REGION Network 2: Перше слово повідомлень
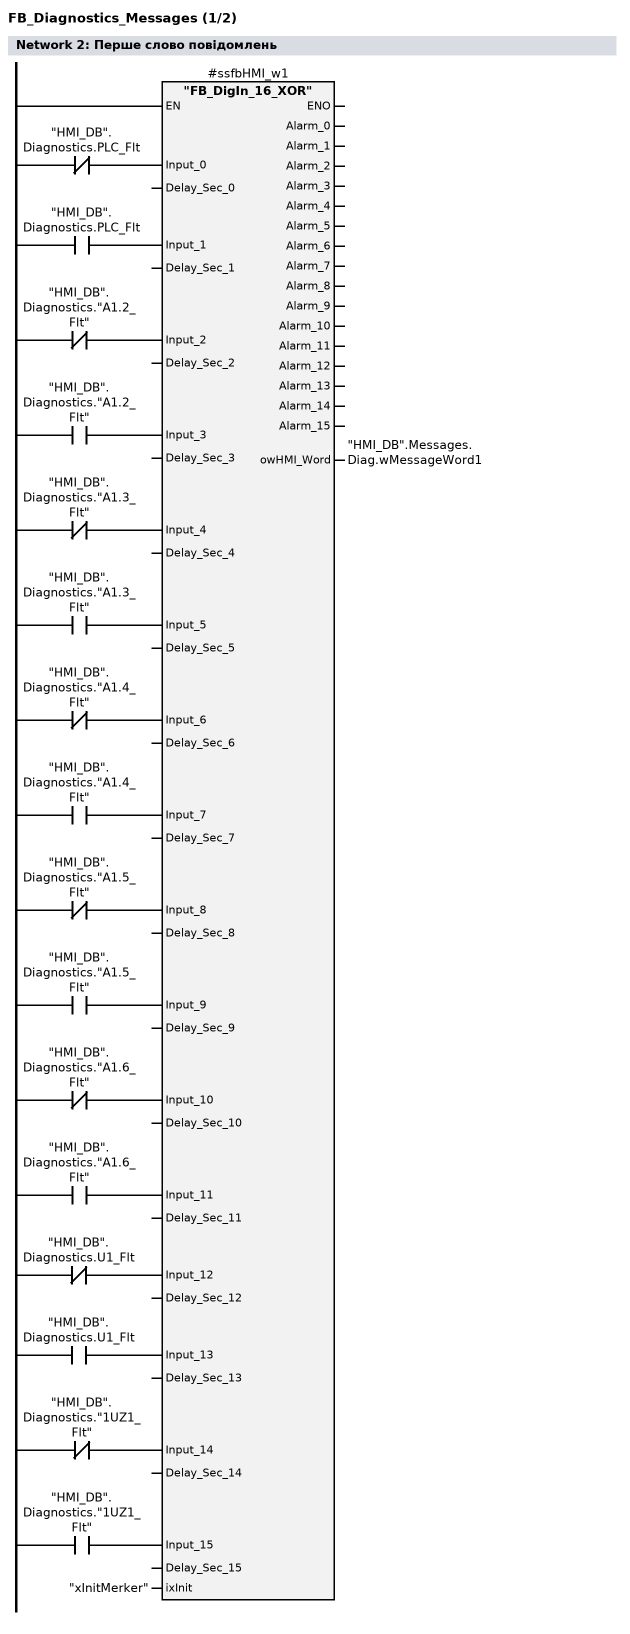
   RUNG wire#powerrail
      #ssfbHMI_w1(Input_0 := wire#w1, Input_1 := wire#w2, Input_2 := wire#w3, Input_3 := wire#w4, Input_4 := wire#w5, Input_5 := wire#w6, Input_6 := wire#w7, Input_7 := wire#w8, Input_8 := wire#w9, Input_9 := wire#w10, Input_10 := wire#w11, Input_11 := wire#w12, Input_12 := wire#w13, Input_13 := wire#w14, Input_14 := wire#w15, Input_15 := wire#w16, Delay_Sec_0 :=, Delay_Sec_1 :=, Delay_Sec_2 :=, Delay_Sec_3 :=, Delay_Sec_4 :=, Delay_Sec_5 :=, Delay_Sec_6 :=, Delay_Sec_7 :=, Delay_Sec_8 :=, Delay_Sec_9 :=, Delay_Sec_10 :=, Delay_Sec_11 :=, Delay_Sec_12 :=, Delay_Sec_13 :=, Delay_Sec_14 :=, Delay_Sec_15 :=, ixInit := "xInitMerker", Alarm_0 =>, Alarm_1 =>, Alarm_2 =>, Alarm_3 =>, Alarm_4 =>, Alarm_5 =>, Alarm_6 =>, Alarm_7 =>, Alarm_8 =>, Alarm_9 =>, Alarm_10 =>, Alarm_11 =>, Alarm_12 =>, Alarm_13 =>, Alarm_14 =>, Alarm_15 =>, owHMI_Word => "HMI_DB".Messages.Diag.wMessageWord1)
   END_RUNG
   RUNG wire#powerrail
      I_Contact( "HMI_DB".Diagnostics.PLC_Flt )
   END_RUNG wire#w1
   RUNG wire#powerrail
      Contact( "HMI_DB".Diagnostics.PLC_Flt )
   END_RUNG wire#w2
   RUNG wire#powerrail
      I_Contact( "HMI_DB".Diagnostics."A1.2_Flt" )
   END_RUNG wire#w3
   RUNG wire#powerrail
      Contact( "HMI_DB".Diagnostics."A1.2_Flt" )
   END_RUNG wire#w4
   RUNG wire#powerrail
      I_Contact( "HMI_DB".Diagnostics."A1.3_Flt" )
   END_RUNG wire#w5
   RUNG wire#powerrail
      Contact( "HMI_DB".Diagnostics."A1.3_Flt" )
   END_RUNG wire#w6
   RUNG wire#powerrail
      I_Contact( "HMI_DB".Diagnostics."A1.4_Flt" )
   END_RUNG wire#w7
   RUNG wire#powerrail
      Contact( "HMI_DB".Diagnostics."A1.4_Flt" )
   END_RUNG wire#w8
   RUNG wire#powerrail
      I_Contact( "HMI_DB".Diagnostics."A1.5_Flt" )
   END_RUNG wire#w9
   RUNG wire#powerrail
      Contact( "HMI_DB".Diagnostics."A1.5_Flt" )
   END_RUNG wire#w10
   RUNG wire#powerrail
      I_Contact( "HMI_DB".Diagnostics."A1.6_Flt" )
   END_RUNG wire#w11
   RUNG wire#powerrail
      Contact( "HMI_DB".Diagnostics."A1.6_Flt" )
   END_RUNG wire#w12
   RUNG wire#powerrail
      I_Contact( "HMI_DB".Diagnostics.U1_Flt )
   END_RUNG wire#w13
   RUNG wire#powerrail
      Contact( "HMI_DB".Diagnostics.U1_Flt )
   END_RUNG wire#w14
   RUNG wire#powerrail
      I_Contact( "HMI_DB".Diagnostics."1UZ1_Flt" )
   END_RUNG wire#w15
   RUNG wire#powerrail
      Contact( "HMI_DB".Diagnostics."1UZ1_Flt" )
   END_RUNG wire#w16
   // the same network as SCL:
   #ssfbHMI_w1(Input_0 := NOT "HMI_DB".Diagnostics.PLC_Flt,   // "FB_DigIn_16_XOR"
               Input_1 := "HMI_DB".Diagnostics.PLC_Flt,
               Input_2 := NOT "HMI_DB".Diagnostics."A1.2_Flt",
               Input_3 := "HMI_DB".Diagnostics."A1.2_Flt",
               Input_4 := NOT "HMI_DB".Diagnostics."A1.3_Flt",
               Input_5 := "HMI_DB".Diagnostics."A1.3_Flt",
               Input_6 := NOT "HMI_DB".Diagnostics."A1.4_Flt",
               Input_7 := "HMI_DB".Diagnostics."A1.4_Flt",
               Input_8 := NOT "HMI_DB".Diagnostics."A1.5_Flt",
               Input_9 := "HMI_DB".Diagnostics."A1.5_Flt",
               Input_10 := NOT "HMI_DB".Diagnostics."A1.6_Flt",
               Input_11 := "HMI_DB".Diagnostics."A1.6_Flt",
               Input_12 := NOT "HMI_DB".Diagnostics.U1_Flt,
               Input_13 := "HMI_DB".Diagnostics.U1_Flt,
               Input_14 := NOT "HMI_DB".Diagnostics."1UZ1_Flt",
               Input_15 := "HMI_DB".Diagnostics."1UZ1_Flt",
               ixInit := "xInitMerker",
               owHMI_Word => "HMI_DB".Messages.Diag.wMessageWord1);
END_REGION

REGION Network 3: Друге слово повідомлень
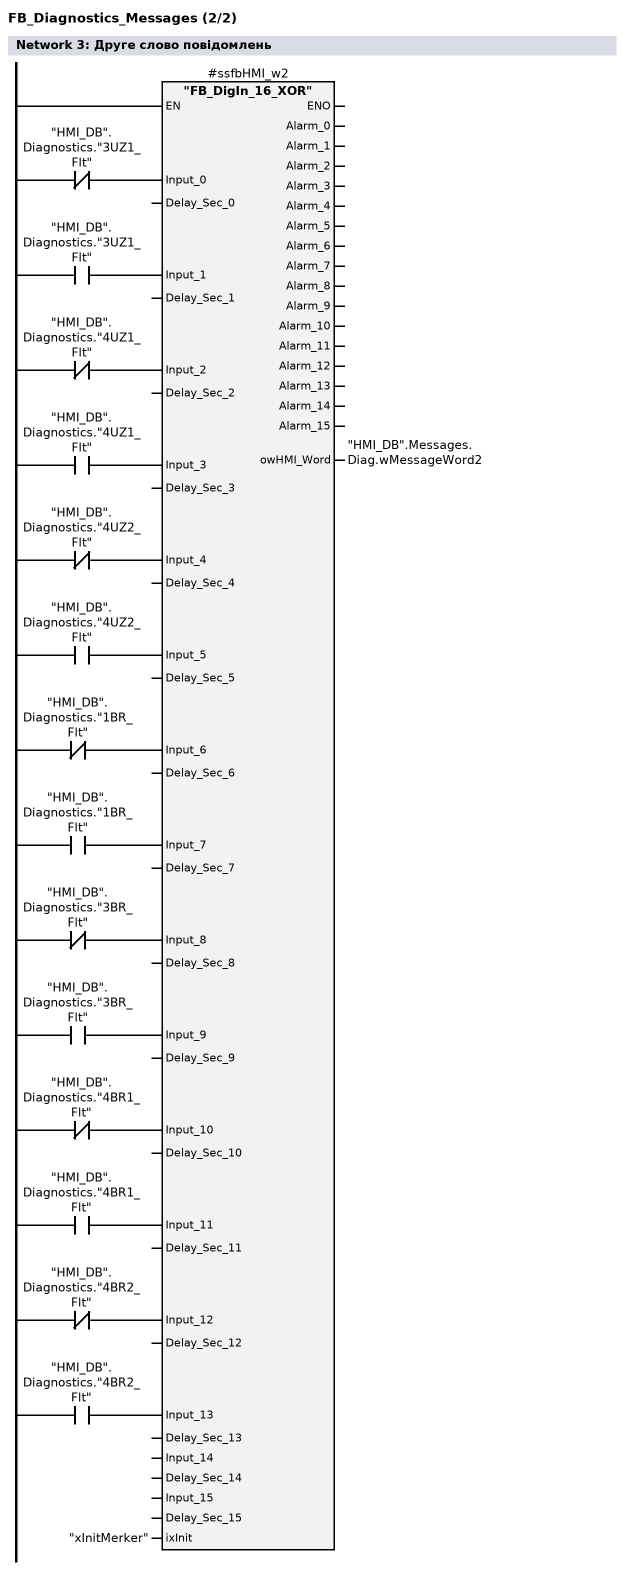
   RUNG wire#powerrail
      #ssfbHMI_w2(Input_0 := wire#w1, Input_1 := wire#w2, Input_2 := wire#w3, Input_3 := wire#w4, Input_4 := wire#w5, Input_5 := wire#w6, Input_6 := wire#w7, Input_7 := wire#w8, Input_8 := wire#w9, Input_9 := wire#w10, Input_10 := wire#w11, Input_11 := wire#w12, Input_12 := wire#w13, Input_13 := wire#w14, Delay_Sec_0 :=, Delay_Sec_1 :=, Delay_Sec_2 :=, Delay_Sec_3 :=, Delay_Sec_4 :=, Delay_Sec_5 :=, Delay_Sec_6 :=, Delay_Sec_7 :=, Delay_Sec_8 :=, Delay_Sec_9 :=, Delay_Sec_10 :=, Delay_Sec_11 :=, Delay_Sec_12 :=, Delay_Sec_13 :=, Input_14 :=, Delay_Sec_14 :=, Input_15 :=, Delay_Sec_15 :=, ixInit := "xInitMerker", Alarm_0 =>, Alarm_1 =>, Alarm_2 =>, Alarm_3 =>, Alarm_4 =>, Alarm_5 =>, Alarm_6 =>, Alarm_7 =>, Alarm_8 =>, Alarm_9 =>, Alarm_10 =>, Alarm_11 =>, Alarm_12 =>, Alarm_13 =>, Alarm_14 =>, Alarm_15 =>, owHMI_Word => "HMI_DB".Messages.Diag.wMessageWord2)
   END_RUNG
   RUNG wire#powerrail
      I_Contact( "HMI_DB".Diagnostics."3UZ1_Flt" )
   END_RUNG wire#w1
   RUNG wire#powerrail
      Contact( "HMI_DB".Diagnostics."3UZ1_Flt" )
   END_RUNG wire#w2
   RUNG wire#powerrail
      I_Contact( "HMI_DB".Diagnostics."4UZ1_Flt" )
   END_RUNG wire#w3
   RUNG wire#powerrail
      Contact( "HMI_DB".Diagnostics."4UZ1_Flt" )
   END_RUNG wire#w4
   RUNG wire#powerrail
      I_Contact( "HMI_DB".Diagnostics."4UZ2_Flt" )
   END_RUNG wire#w5
   RUNG wire#powerrail
      Contact( "HMI_DB".Diagnostics."4UZ2_Flt" )
   END_RUNG wire#w6
   RUNG wire#powerrail
      I_Contact( "HMI_DB".Diagnostics."1BR_Flt" )
   END_RUNG wire#w7
   RUNG wire#powerrail
      Contact( "HMI_DB".Diagnostics."1BR_Flt" )
   END_RUNG wire#w8
   RUNG wire#powerrail
      I_Contact( "HMI_DB".Diagnostics."3BR_Flt" )
   END_RUNG wire#w9
   RUNG wire#powerrail
      Contact( "HMI_DB".Diagnostics."3BR_Flt" )
   END_RUNG wire#w10
   RUNG wire#powerrail
      I_Contact( "HMI_DB".Diagnostics."4BR1_Flt" )
   END_RUNG wire#w11
   RUNG wire#powerrail
      Contact( "HMI_DB".Diagnostics."4BR1_Flt" )
   END_RUNG wire#w12
   RUNG wire#powerrail
      I_Contact( "HMI_DB".Diagnostics."4BR2_Flt" )
   END_RUNG wire#w13
   RUNG wire#powerrail
      Contact( "HMI_DB".Diagnostics."4BR2_Flt" )
   END_RUNG wire#w14
   // the same network as SCL:
   #ssfbHMI_w2(Input_0 := NOT "HMI_DB".Diagnostics."3UZ1_Flt",   // "FB_DigIn_16_XOR"
               Input_1 := "HMI_DB".Diagnostics."3UZ1_Flt",
               Input_2 := NOT "HMI_DB".Diagnostics."4UZ1_Flt",
               Input_3 := "HMI_DB".Diagnostics."4UZ1_Flt",
               Input_4 := NOT "HMI_DB".Diagnostics."4UZ2_Flt",
               Input_5 := "HMI_DB".Diagnostics."4UZ2_Flt",
               Input_6 := NOT "HMI_DB".Diagnostics."1BR_Flt",
               Input_7 := "HMI_DB".Diagnostics."1BR_Flt",
               Input_8 := NOT "HMI_DB".Diagnostics."3BR_Flt",
               Input_9 := "HMI_DB".Diagnostics."3BR_Flt",
               Input_10 := NOT "HMI_DB".Diagnostics."4BR1_Flt",
               Input_11 := "HMI_DB".Diagnostics."4BR1_Flt",
               Input_12 := NOT "HMI_DB".Diagnostics."4BR2_Flt",
               Input_13 := "HMI_DB".Diagnostics."4BR2_Flt",
               ixInit := "xInitMerker",
               owHMI_Word => "HMI_DB".Messages.Diag.wMessageWord2);
END_REGION
END_FUNCTION_BLOCK

FUNCTION "FC_Diagnostic" : Void   // FC600, LAD
{ S7_Optimized_Access := 'TRUE' }
VERSION : 0.1
BEGIN

REGION Network 2: =================ПЛК=======================
END_REGION

REGION Network 3: CPU 1515-2 PN
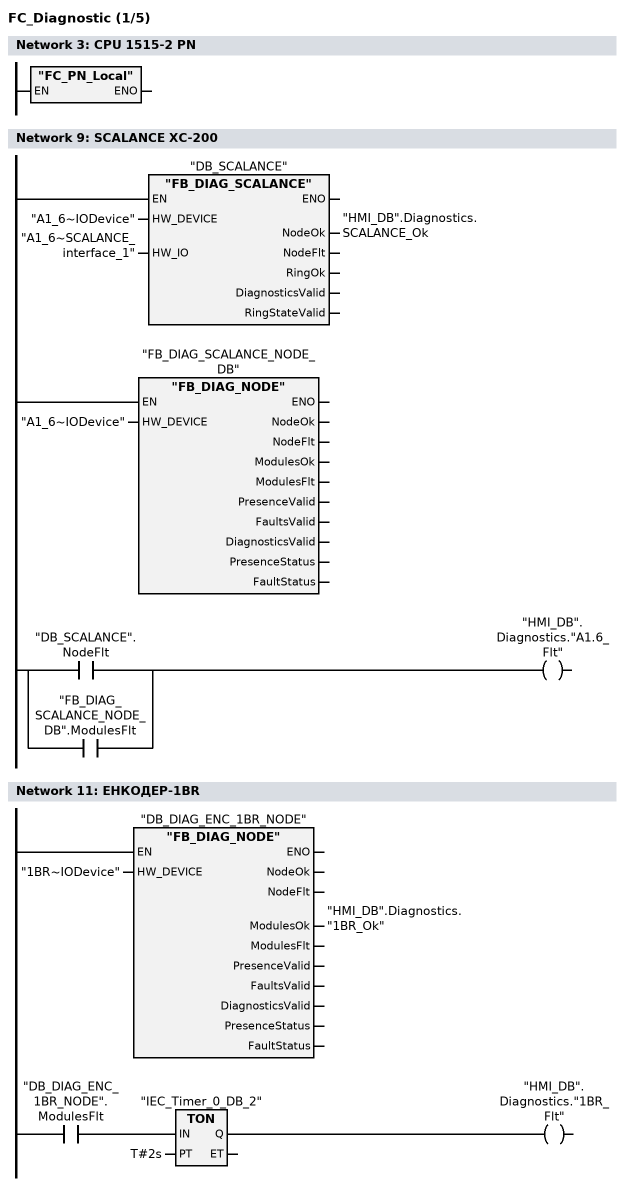
   RUNG wire#powerrail
      "FC_PN_Local"()
   END_RUNG
   // the same network as SCL:
   "FC_PN_Local"();
END_REGION

REGION Network 4: Модуль А1.2
END_REGION

REGION Network 5: Модуль А1.3
END_REGION

REGION Network 6: Модуль А1.4
END_REGION

REGION Network 7: Модуль А1.5
END_REGION

REGION Network 8: =================Мережева діагностіка=======================
END_REGION

REGION Network 9: SCALANCE XC-200
   RUNG wire#powerrail
      "DB_SCALANCE"(HW_DEVICE := "A1_6~IODevice", HW_IO := "A1_6~SCALANCE_interface_1", NodeOk => "HMI_DB".Diagnostics.SCALANCE_Ok, NodeFlt =>, RingOk =>, DiagnosticsValid =>, RingStateValid =>)
   END_RUNG
   RUNG wire#powerrail
      "FB_DIAG_SCALANCE_NODE_DB"(HW_DEVICE := "A1_6~IODevice", NodeOk =>, NodeFlt =>, ModulesOk =>, ModulesFlt =>, PresenceValid =>, FaultsValid =>, DiagnosticsValid =>, PresenceStatus =>, FaultStatus =>)
   END_RUNG
   RUNG wire#powerrail
      Contact( "DB_SCALANCE".NodeFlt )
      wire#w1
      Coil( "HMI_DB".Diagnostics."A1.6_Flt" )
   END_RUNG
   RUNG wire#powerrail
      Contact( "FB_DIAG_SCALANCE_NODE_DB".ModulesFlt )
   END_RUNG wire#w1
   // the same network as SCL:
   "DB_SCALANCE"(HW_DEVICE := "A1_6~IODevice",   // "FB_DIAG_SCALANCE"
                 HW_IO := "A1_6~SCALANCE_interface_1",
                 NodeOk => "HMI_DB".Diagnostics.SCALANCE_Ok);
   "FB_DIAG_SCALANCE_NODE_DB"(HW_DEVICE := "A1_6~IODevice");   // "FB_DIAG_NODE"
   "HMI_DB".Diagnostics."A1.6_Flt" := "DB_SCALANCE".NodeFlt OR "FB_DIAG_SCALANCE_NODE_DB".ModulesFlt;
END_REGION

REGION Network 10: =================Енкодери==================
END_REGION

REGION Network 11: ЕНКОДЕР-1BR
   "DB_DIAG_ENC_1BR_NODE"(HW_DEVICE := "1BR~IODevice", ModulesOk => "HMI_DB".Diagnostics."1BR_Ok");   // "FB_DIAG_NODE"
   "IEC_Timer_0_DB_2".TON(IN := "DB_DIAG_ENC_1BR_NODE".ModulesFlt, PT := T#2s);
   "HMI_DB".Diagnostics."1BR_Flt" := "IEC_Timer_0_DB_2".Q;
END_REGION

REGION Network 12: ЕНКОДЕР-3BR
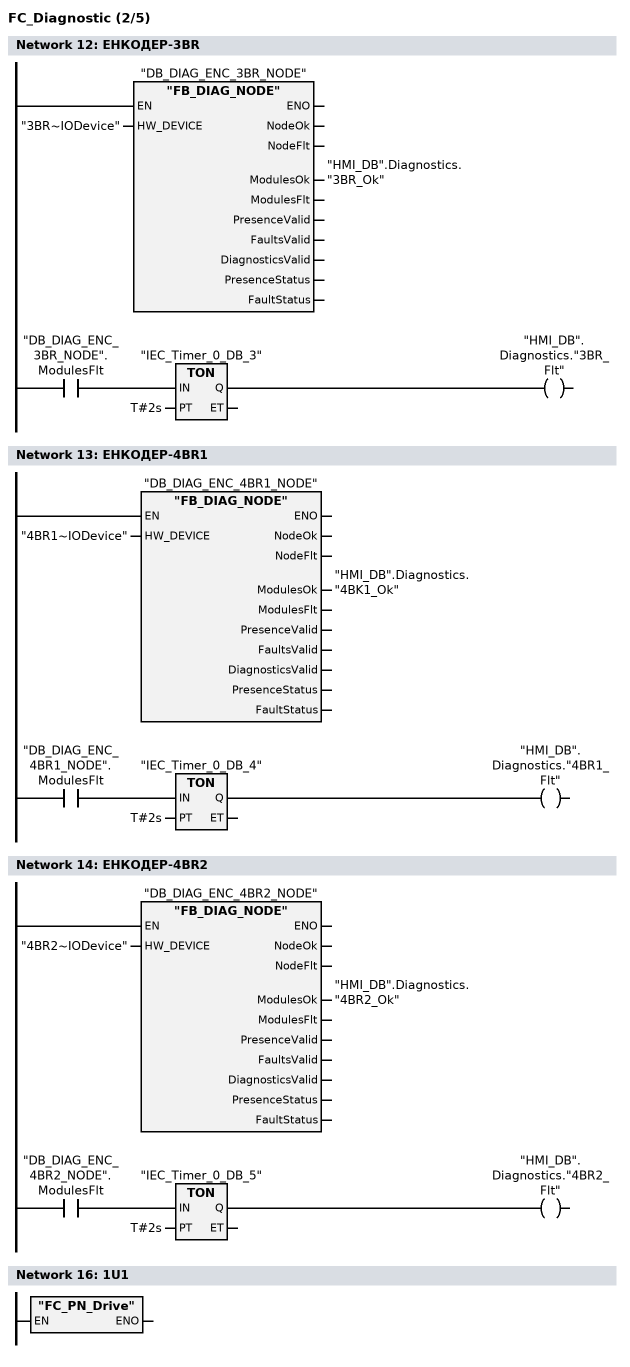
   "DB_DIAG_ENC_3BR_NODE"(HW_DEVICE := "3BR~IODevice", ModulesOk => "HMI_DB".Diagnostics."3BR_Ok");   // "FB_DIAG_NODE"
   "IEC_Timer_0_DB_3".TON(IN := "DB_DIAG_ENC_3BR_NODE".ModulesFlt, PT := T#2s);
   "HMI_DB".Diagnostics."3BR_Flt" := "IEC_Timer_0_DB_3".Q;
END_REGION

REGION Network 13: ЕНКОДЕР-4BR1
   "DB_DIAG_ENC_4BR1_NODE"(HW_DEVICE := "4BR1~IODevice", ModulesOk => "HMI_DB".Diagnostics."4BK1_Ok");   // "FB_DIAG_NODE"
   "IEC_Timer_0_DB_4".TON(IN := "DB_DIAG_ENC_4BR1_NODE".ModulesFlt, PT := T#2s);
   "HMI_DB".Diagnostics."4BR1_Flt" := "IEC_Timer_0_DB_4".Q;
END_REGION

REGION Network 14: ЕНКОДЕР-4BR2
   "DB_DIAG_ENC_4BR2_NODE"(HW_DEVICE := "4BR2~IODevice", ModulesOk => "HMI_DB".Diagnostics."4BR2_Ok");   // "FB_DIAG_NODE"
   "IEC_Timer_0_DB_5".TON(IN := "DB_DIAG_ENC_4BR2_NODE".ModulesFlt, PT := T#2s);
   "HMI_DB".Diagnostics."4BR2_Flt" := "IEC_Timer_0_DB_5".Q;
END_REGION

REGION Network 15: =================ПЧ======================
END_REGION

REGION Network 16: 1U1
   RUNG wire#powerrail
      "FC_PN_Drive"()
   END_RUNG
   // the same network as SCL:
   "FC_PN_Drive"();
END_REGION

REGION Network 17: 1UZ1
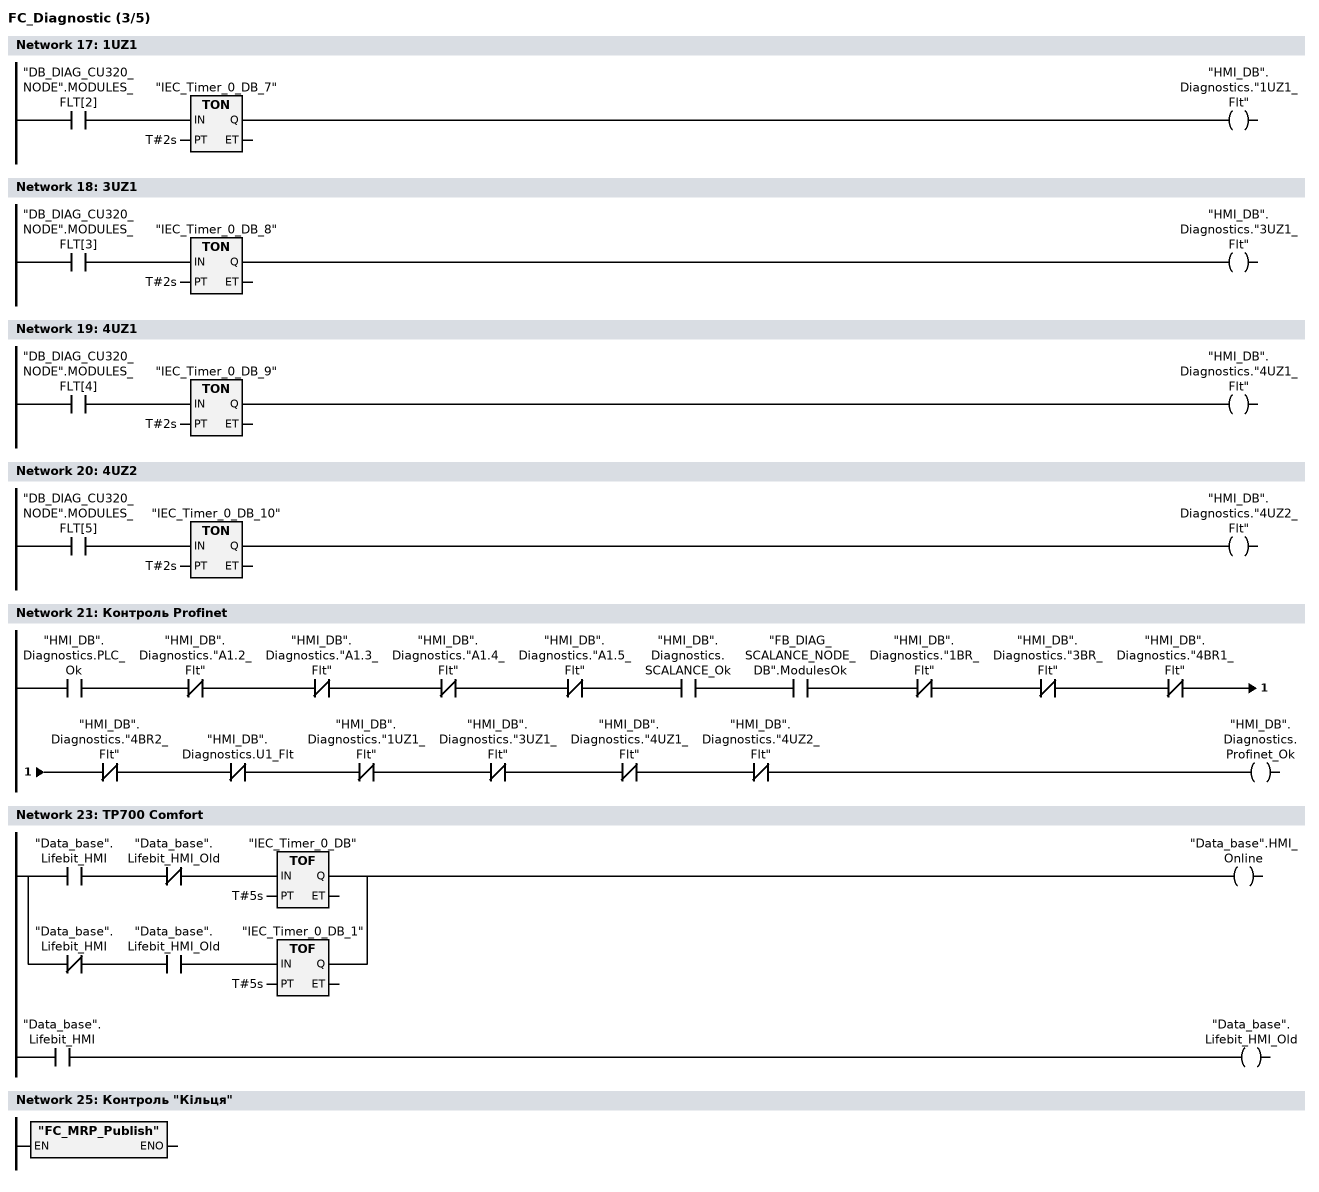
   "IEC_Timer_0_DB_7".TON(IN := "DB_DIAG_CU320_NODE".MODULES_FLT[2], PT := T#2s);
   "HMI_DB".Diagnostics."1UZ1_Flt" := "IEC_Timer_0_DB_7".Q;
END_REGION

REGION Network 18: 3UZ1
   "IEC_Timer_0_DB_8".TON(IN := "DB_DIAG_CU320_NODE".MODULES_FLT[3], PT := T#2s);
   "HMI_DB".Diagnostics."3UZ1_Flt" := "IEC_Timer_0_DB_8".Q;
END_REGION

REGION Network 19: 4UZ1
   "IEC_Timer_0_DB_9".TON(IN := "DB_DIAG_CU320_NODE".MODULES_FLT[4], PT := T#2s);
   "HMI_DB".Diagnostics."4UZ1_Flt" := "IEC_Timer_0_DB_9".Q;
END_REGION

REGION Network 20: 4UZ2
   "IEC_Timer_0_DB_10".TON(IN := "DB_DIAG_CU320_NODE".MODULES_FLT[5], PT := T#2s);
   "HMI_DB".Diagnostics."4UZ2_Flt" := "IEC_Timer_0_DB_10".Q;
END_REGION

REGION Network 21: Контроль Profinet
   RUNG wire#powerrail
      Contact( "HMI_DB".Diagnostics.PLC_Ok )
      I_Contact( "HMI_DB".Diagnostics."A1.2_Flt" )
      I_Contact( "HMI_DB".Diagnostics."A1.3_Flt" )
      I_Contact( "HMI_DB".Diagnostics."A1.4_Flt" )
      I_Contact( "HMI_DB".Diagnostics."A1.5_Flt" )
      Contact( "HMI_DB".Diagnostics.SCALANCE_Ok )
      Contact( "FB_DIAG_SCALANCE_NODE_DB".ModulesOk )
      I_Contact( "HMI_DB".Diagnostics."1BR_Flt" )
      I_Contact( "HMI_DB".Diagnostics."3BR_Flt" )
      I_Contact( "HMI_DB".Diagnostics."4BR1_Flt" )
      I_Contact( "HMI_DB".Diagnostics."4BR2_Flt" )
      I_Contact( "HMI_DB".Diagnostics.U1_Flt )
      I_Contact( "HMI_DB".Diagnostics."1UZ1_Flt" )
      I_Contact( "HMI_DB".Diagnostics."3UZ1_Flt" )
      I_Contact( "HMI_DB".Diagnostics."4UZ1_Flt" )
      I_Contact( "HMI_DB".Diagnostics."4UZ2_Flt" )
      Coil( "HMI_DB".Diagnostics.Profinet_Ok )
   END_RUNG
   // the same network as SCL:
   "HMI_DB".Diagnostics.Profinet_Ok := "HMI_DB".Diagnostics.PLC_Ok AND NOT "HMI_DB".Diagnostics."A1.2_Flt" AND NOT "HMI_DB".Diagnostics."A1.3_Flt" AND NOT "HMI_DB".Diagnostics."A1.4_Flt" AND NOT "HMI_DB".Diagnostics."A1.5_Flt" AND "HMI_DB".Diagnostics.SCALANCE_Ok AND "FB_DIAG_SCALANCE_NODE_DB".ModulesOk AND NOT "HMI_DB".Diagnostics."1BR_Flt" AND NOT "HMI_DB".Diagnostics."3BR_Flt" AND NOT "HMI_DB".Diagnostics."4BR1_Flt" AND NOT "HMI_DB".Diagnostics."4BR2_Flt" AND NOT "HMI_DB".Diagnostics.U1_Flt AND NOT "HMI_DB".Diagnostics."1UZ1_Flt" AND NOT "HMI_DB".Diagnostics."3UZ1_Flt" AND NOT "HMI_DB".Diagnostics."4UZ1_Flt" AND NOT "HMI_DB".Diagnostics."4UZ2_Flt";
END_REGION

REGION Network 22: ================ЛMI======================
END_REGION

REGION Network 23: TP700 Comfort
   "IEC_Timer_0_DB".TOF(IN := "Data_base".Lifebit_HMI AND NOT "Data_base".Lifebit_HMI_Old, PT := T#5s);
   "IEC_Timer_0_DB_1".TOF(IN := NOT "Data_base".Lifebit_HMI AND "Data_base".Lifebit_HMI_Old, PT := T#5s);
   "Data_base".HMI_Online := "IEC_Timer_0_DB".Q OR "IEC_Timer_0_DB_1".Q;
   "Data_base".Lifebit_HMI_Old := "Data_base".Lifebit_HMI;
END_REGION

REGION Network 24: =========================================
END_REGION

REGION Network 25: Контроль "Кільця"
   RUNG wire#powerrail
      "FC_MRP_Publish"()
   END_RUNG
   // the same network as SCL:
   "FC_MRP_Publish"();
END_REGION

REGION Network 26: Формування слова аварій
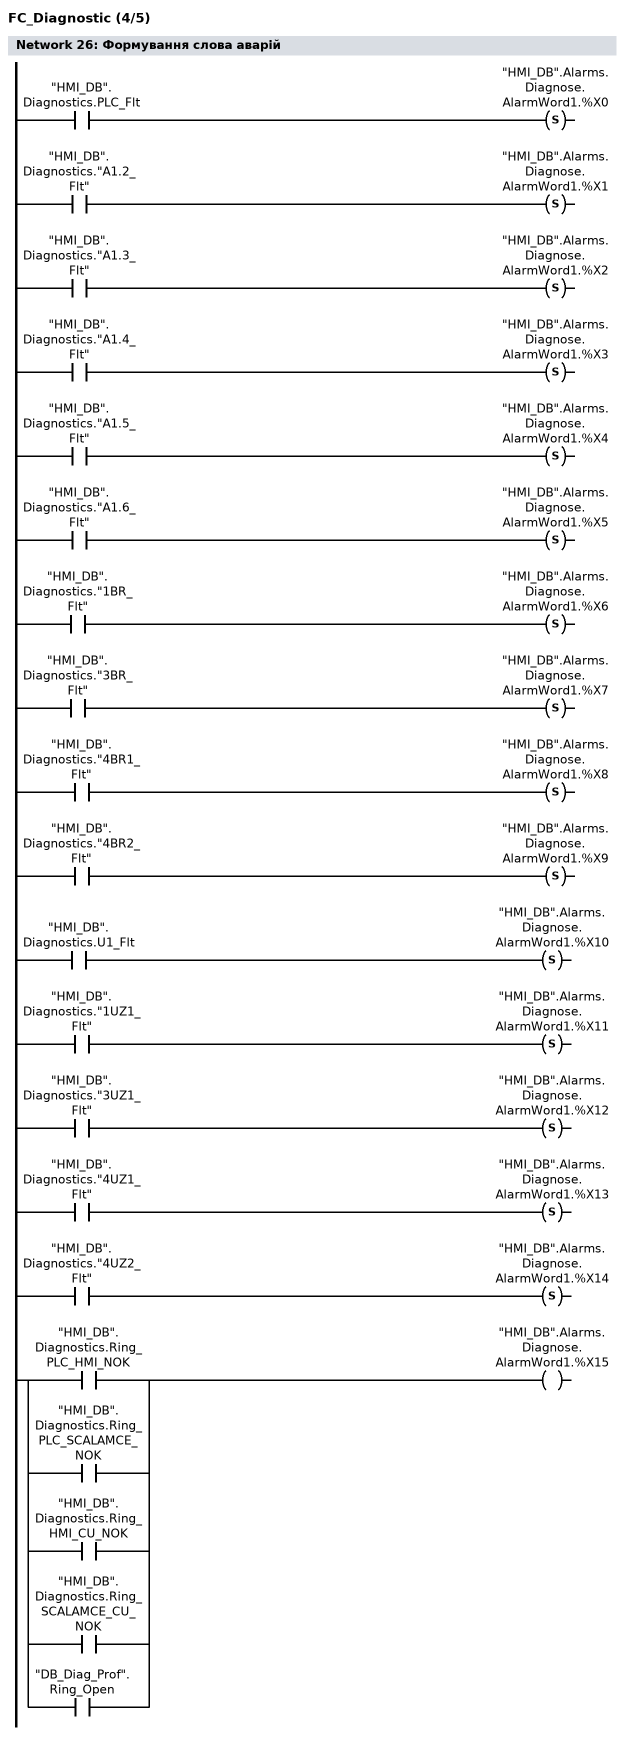
   RUNG wire#powerrail
      Contact( "HMI_DB".Diagnostics.PLC_Flt )
      S_Coil( "HMI_DB".Alarms.Diagnose.AlarmWord1.%X0 )
   END_RUNG
   RUNG wire#powerrail
      Contact( "HMI_DB".Diagnostics."A1.2_Flt" )
      S_Coil( "HMI_DB".Alarms.Diagnose.AlarmWord1.%X1 )
   END_RUNG
   RUNG wire#powerrail
      Contact( "HMI_DB".Diagnostics."A1.3_Flt" )
      S_Coil( "HMI_DB".Alarms.Diagnose.AlarmWord1.%X2 )
   END_RUNG
   RUNG wire#powerrail
      Contact( "HMI_DB".Diagnostics."A1.4_Flt" )
      S_Coil( "HMI_DB".Alarms.Diagnose.AlarmWord1.%X3 )
   END_RUNG
   RUNG wire#powerrail
      Contact( "HMI_DB".Diagnostics."A1.5_Flt" )
      S_Coil( "HMI_DB".Alarms.Diagnose.AlarmWord1.%X4 )
   END_RUNG
   RUNG wire#powerrail
      Contact( "HMI_DB".Diagnostics."A1.6_Flt" )
      S_Coil( "HMI_DB".Alarms.Diagnose.AlarmWord1.%X5 )
   END_RUNG
   RUNG wire#powerrail
      Contact( "HMI_DB".Diagnostics."1BR_Flt" )
      S_Coil( "HMI_DB".Alarms.Diagnose.AlarmWord1.%X6 )
   END_RUNG
   RUNG wire#powerrail
      Contact( "HMI_DB".Diagnostics."3BR_Flt" )
      S_Coil( "HMI_DB".Alarms.Diagnose.AlarmWord1.%X7 )
   END_RUNG
   RUNG wire#powerrail
      Contact( "HMI_DB".Diagnostics."4BR1_Flt" )
      S_Coil( "HMI_DB".Alarms.Diagnose.AlarmWord1.%X8 )
   END_RUNG
   RUNG wire#powerrail
      Contact( "HMI_DB".Diagnostics."4BR2_Flt" )
      S_Coil( "HMI_DB".Alarms.Diagnose.AlarmWord1.%X9 )
   END_RUNG
   RUNG wire#powerrail
      Contact( "HMI_DB".Diagnostics.U1_Flt )
      S_Coil( "HMI_DB".Alarms.Diagnose.AlarmWord1.%X10 )
   END_RUNG
   RUNG wire#powerrail
      Contact( "HMI_DB".Diagnostics."1UZ1_Flt" )
      S_Coil( "HMI_DB".Alarms.Diagnose.AlarmWord1.%X11 )
   END_RUNG
   RUNG wire#powerrail
      Contact( "HMI_DB".Diagnostics."3UZ1_Flt" )
      S_Coil( "HMI_DB".Alarms.Diagnose.AlarmWord1.%X12 )
   END_RUNG
   RUNG wire#powerrail
      Contact( "HMI_DB".Diagnostics."4UZ1_Flt" )
      S_Coil( "HMI_DB".Alarms.Diagnose.AlarmWord1.%X13 )
   END_RUNG
   RUNG wire#powerrail
      Contact( "HMI_DB".Diagnostics."4UZ2_Flt" )
      S_Coil( "HMI_DB".Alarms.Diagnose.AlarmWord1.%X14 )
   END_RUNG
   RUNG wire#powerrail
      Contact( "HMI_DB".Diagnostics.Ring_PLC_HMI_NOK )
      wire#w1
      Coil( "HMI_DB".Alarms.Diagnose.AlarmWord1.%X15 )
   END_RUNG
   RUNG wire#powerrail
      Contact( "HMI_DB".Diagnostics.Ring_PLC_SCALAMCE_NOK )
   END_RUNG wire#w1
   RUNG wire#powerrail
      Contact( "HMI_DB".Diagnostics.Ring_HMI_CU_NOK )
   END_RUNG wire#w1
   RUNG wire#powerrail
      Contact( "HMI_DB".Diagnostics.Ring_SCALAMCE_CU_NOK )
   END_RUNG wire#w1
   RUNG wire#powerrail
      Contact( "DB_Diag_Prof".Ring_Open )
   END_RUNG wire#w1
   // the same network as SCL:
   IF "HMI_DB".Diagnostics.PLC_Flt THEN "HMI_DB".Alarms.Diagnose.AlarmWord1.%X0 := TRUE; END_IF;
   IF "HMI_DB".Diagnostics."A1.2_Flt" THEN "HMI_DB".Alarms.Diagnose.AlarmWord1.%X1 := TRUE; END_IF;
   IF "HMI_DB".Diagnostics."A1.3_Flt" THEN "HMI_DB".Alarms.Diagnose.AlarmWord1.%X2 := TRUE; END_IF;
   IF "HMI_DB".Diagnostics."A1.4_Flt" THEN "HMI_DB".Alarms.Diagnose.AlarmWord1.%X3 := TRUE; END_IF;
   IF "HMI_DB".Diagnostics."A1.5_Flt" THEN "HMI_DB".Alarms.Diagnose.AlarmWord1.%X4 := TRUE; END_IF;
   IF "HMI_DB".Diagnostics."A1.6_Flt" THEN "HMI_DB".Alarms.Diagnose.AlarmWord1.%X5 := TRUE; END_IF;
   IF "HMI_DB".Diagnostics."1BR_Flt" THEN "HMI_DB".Alarms.Diagnose.AlarmWord1.%X6 := TRUE; END_IF;
   IF "HMI_DB".Diagnostics."3BR_Flt" THEN "HMI_DB".Alarms.Diagnose.AlarmWord1.%X7 := TRUE; END_IF;
   IF "HMI_DB".Diagnostics."4BR1_Flt" THEN "HMI_DB".Alarms.Diagnose.AlarmWord1.%X8 := TRUE; END_IF;
   IF "HMI_DB".Diagnostics."4BR2_Flt" THEN "HMI_DB".Alarms.Diagnose.AlarmWord1.%X9 := TRUE; END_IF;
   IF "HMI_DB".Diagnostics.U1_Flt THEN "HMI_DB".Alarms.Diagnose.AlarmWord1.%X10 := TRUE; END_IF;
   IF "HMI_DB".Diagnostics."1UZ1_Flt" THEN "HMI_DB".Alarms.Diagnose.AlarmWord1.%X11 := TRUE; END_IF;
   IF "HMI_DB".Diagnostics."3UZ1_Flt" THEN "HMI_DB".Alarms.Diagnose.AlarmWord1.%X12 := TRUE; END_IF;
   IF "HMI_DB".Diagnostics."4UZ1_Flt" THEN "HMI_DB".Alarms.Diagnose.AlarmWord1.%X13 := TRUE; END_IF;
   IF "HMI_DB".Diagnostics."4UZ2_Flt" THEN "HMI_DB".Alarms.Diagnose.AlarmWord1.%X14 := TRUE; END_IF;
   "HMI_DB".Alarms.Diagnose.AlarmWord1.%X15 := "HMI_DB".Diagnostics.Ring_PLC_HMI_NOK OR "HMI_DB".Diagnostics.Ring_PLC_SCALAMCE_NOK OR "HMI_DB".Diagnostics.Ring_HMI_CU_NOK OR "HMI_DB".Diagnostics.Ring_SCALAMCE_CU_NOK OR "DB_Diag_Prof".Ring_Open;
END_REGION

REGION Network 27: Скидання слова аварій
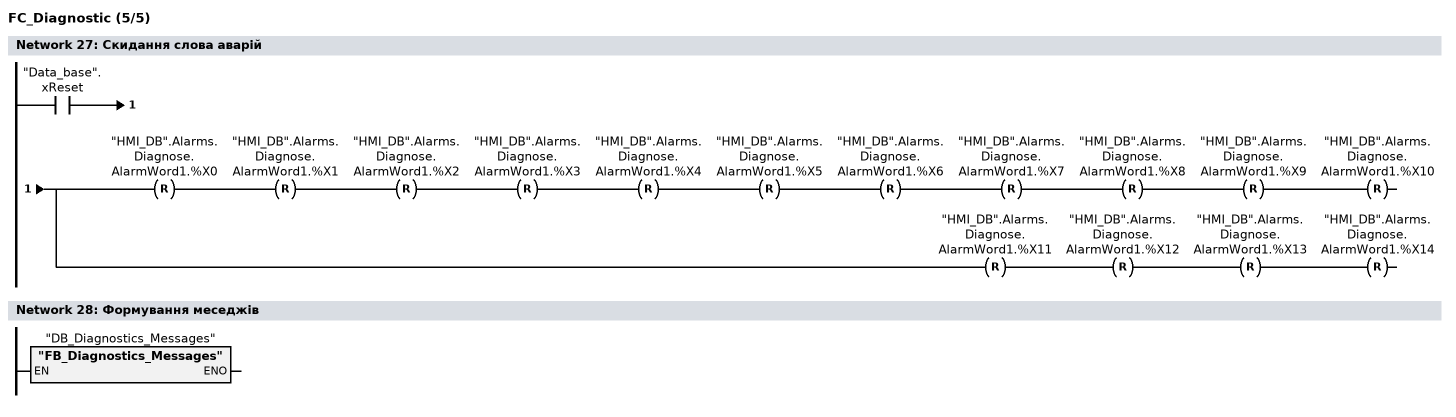
   RUNG wire#powerrail
      Contact( "Data_base".xReset )
      wire#w1
      R_Coil( "HMI_DB".Alarms.Diagnose.AlarmWord1.%X0 )
      R_Coil( "HMI_DB".Alarms.Diagnose.AlarmWord1.%X1 )
      R_Coil( "HMI_DB".Alarms.Diagnose.AlarmWord1.%X2 )
      R_Coil( "HMI_DB".Alarms.Diagnose.AlarmWord1.%X3 )
      R_Coil( "HMI_DB".Alarms.Diagnose.AlarmWord1.%X4 )
      R_Coil( "HMI_DB".Alarms.Diagnose.AlarmWord1.%X5 )
      R_Coil( "HMI_DB".Alarms.Diagnose.AlarmWord1.%X6 )
      R_Coil( "HMI_DB".Alarms.Diagnose.AlarmWord1.%X7 )
      R_Coil( "HMI_DB".Alarms.Diagnose.AlarmWord1.%X8 )
      R_Coil( "HMI_DB".Alarms.Diagnose.AlarmWord1.%X9 )
      R_Coil( "HMI_DB".Alarms.Diagnose.AlarmWord1.%X10 )
   END_RUNG
   RUNG wire#w1
      R_Coil( "HMI_DB".Alarms.Diagnose.AlarmWord1.%X11 )
      R_Coil( "HMI_DB".Alarms.Diagnose.AlarmWord1.%X12 )
      R_Coil( "HMI_DB".Alarms.Diagnose.AlarmWord1.%X13 )
      R_Coil( "HMI_DB".Alarms.Diagnose.AlarmWord1.%X14 )
   END_RUNG
   // the same network as SCL:
   IF "Data_base".xReset THEN
       "HMI_DB".Alarms.Diagnose.AlarmWord1.%X0 := FALSE;
       "HMI_DB".Alarms.Diagnose.AlarmWord1.%X1 := FALSE;
       "HMI_DB".Alarms.Diagnose.AlarmWord1.%X2 := FALSE;
       "HMI_DB".Alarms.Diagnose.AlarmWord1.%X3 := FALSE;
       "HMI_DB".Alarms.Diagnose.AlarmWord1.%X4 := FALSE;
       "HMI_DB".Alarms.Diagnose.AlarmWord1.%X5 := FALSE;
       "HMI_DB".Alarms.Diagnose.AlarmWord1.%X6 := FALSE;
       "HMI_DB".Alarms.Diagnose.AlarmWord1.%X7 := FALSE;
       "HMI_DB".Alarms.Diagnose.AlarmWord1.%X8 := FALSE;
       "HMI_DB".Alarms.Diagnose.AlarmWord1.%X9 := FALSE;
       "HMI_DB".Alarms.Diagnose.AlarmWord1.%X10 := FALSE;
       "HMI_DB".Alarms.Diagnose.AlarmWord1.%X11 := FALSE;
       "HMI_DB".Alarms.Diagnose.AlarmWord1.%X12 := FALSE;
       "HMI_DB".Alarms.Diagnose.AlarmWord1.%X13 := FALSE;
       "HMI_DB".Alarms.Diagnose.AlarmWord1.%X14 := FALSE;
   END_IF;
END_REGION

REGION Network 28: Формування меседжів
   RUNG wire#powerrail
      "DB_Diagnostics_Messages"()
   END_RUNG
   // the same network as SCL:
   "DB_Diagnostics_Messages"();   // "FB_Diagnostics_Messages"
END_REGION
END_FUNCTION

FUNCTION "FC_PN_Local" : Void   // FC610, SCL
{ S7_Optimized_Access := 'TRUE' }
VERSION : 1.0
// FC610. Діагностика локальної станції ПЛК. Оновлює DB_DIAG_NODE, перевіряє достовірність даних та стан модулів у слотах 2–5. Записує наявні ознаки справності й несправності в HMI_DB. Викликається циклічно з мережі 3 FC_Diagnostic.
   VAR_TEMP
      i : Int;   // Індекс циклу обробки елементів.
   END_VAR
BEGIN
   // FC610. Діагностика локальної станції ПЛК. Оновлює DB_DIAG_NODE, перевіряє достовірність даних та стан модулів у слотах 2–5. Записує наявні ознаки справності й несправності в HMI_DB. Викликається циклічно з мережі 3 FC_Diagnostic.
   // Оновлення діагностики локальної станції перед перевіркою її модулів.
   // Індекс -1 у MODULES_FLT є зведеним бітом; індекс n відповідає слоту n.
   // За недостовірних даних модуль не позначається справним. Це впливає на наявні дозволи роботи.

       "DB_DIAG_NODE"(HW_DEVICE := "Local~Device");
       "HMI_DB".Diagnostics.PLC_Ok := "DB_DIAG_NODE".NodeOk;
       "HMI_DB".Diagnostics.PLC_Flt := "DB_DIAG_NODE".NodeFlt;
       "Data_base".ModulStatus := "DB_DIAG_NODE".FaultStatus;
       FOR #i := 0 TO 127 DO
           "Data_base".Moduls_Err[#i] := "DB_DIAG_NODE".MODULES_FLT[#i - 1];
       END_FOR;
       "HMI_DB".Diagnostics."A1.2_Flt" := NOT "DB_DIAG_NODE".DiagnosticsValid OR
           NOT "DB_DIAG_NODE".MODULES_EXISTS[2] OR "DB_DIAG_NODE".MODULES_FLT[2];
       "HMI_DB".Diagnostics."A1.3_Flt" := NOT "DB_DIAG_NODE".DiagnosticsValid OR
           NOT "DB_DIAG_NODE".MODULES_EXISTS[3] OR "DB_DIAG_NODE".MODULES_FLT[3];
       "HMI_DB".Diagnostics."A1.4_Flt" := NOT "DB_DIAG_NODE".DiagnosticsValid OR
           NOT "DB_DIAG_NODE".MODULES_EXISTS[4] OR "DB_DIAG_NODE".MODULES_FLT[4];
       "HMI_DB".Diagnostics."A1.5_Flt" := NOT "DB_DIAG_NODE".DiagnosticsValid OR
           NOT "DB_DIAG_NODE".MODULES_EXISTS[5] OR "DB_DIAG_NODE".MODULES_FLT[5];
       // Зберегти наявні поля стану світлодіодів для сервісних екранів.
       "HMI_DB".Diagnostics.A1_2_LED_Status := LED(LADDR := 257, LED := UINT#2);
       "HMI_DB".Diagnostics.A1_3_LED_Status := LED(LADDR := 258, LED := UINT#2);
       "HMI_DB".Diagnostics.A1_4_LED_Status := LED(LADDR := 259, LED := UINT#2);
       "HMI_DB".Diagnostics.A1_5_LED_Status := LED(LADDR := 260, LED := UINT#2);
END_FUNCTION

FUNCTION "FC_PN_Drive" : Void   // FC611, SCL
{ S7_Optimized_Access := 'TRUE' }
VERSION : 1.0
// FC611. Діагностика вузла привода CU та його модулів. Використовує DB_DIAG_CU320_NODE і апаратний ідентифікатор IO-пристрою привода. Оновлює ознаки HMI, маску наявності модулів і статус читання. Викликається з мережі 16 FC_Diagnostic.
   VAR_TEMP
      i : Int;   // Індекс циклу обробки елементів.
   END_VAR
BEGIN
   // FC611. Діагностика вузла привода CU та його модулів. Використовує DB_DIAG_CU320_NODE і апаратний ідентифікатор IO-пристрою привода. Оновлює ознаки HMI, маску наявності модулів і статус читання. Викликається з мережі 16 FC_Diagnostic.
   // Стан CU враховує несправності його модулів і достовірність діагностики.
   // PROFINET_Status містить наявність модулів: біт 0 — зведений, біт n — слот n-1.
   // Пізніше FB601 уточнює Drive_Online за наявністю IO-пристрою №1.

       "DB_DIAG_CU320_NODE"(HW_DEVICE := "Drive_unit_1~PROFINET_interface~IODevice");
       "HMI_DB".Diagnostics.CU320_Ok := "DB_DIAG_CU320_NODE".ModulesOk;
       "HMI_DB".Diagnostics.U1_Flt := "DB_DIAG_CU320_NODE".ModulesFlt;
       // Буфер сумісності містить перевірену наявність модулів: біт n відповідає слоту n-1.
       "Data_base".RetVal := "DB_DIAG_CU320_NODE".PresenceStatus;
       FOR #i := 0 TO 127 DO
           "Data_base".PROFINET_Status[#i] := "DB_DIAG_CU320_NODE".MODULES_EXISTS[#i - 1];
       END_FOR;
       "Data_base".Drive_Online := "DB_DIAG_CU320_NODE".NodeOk;
END_FUNCTION

FUNCTION "FC_MRP_DecodePort" : Bool   // FC612, SCL
{ S7_Optimized_Access := 'TRUE' }
VERSION : 1.0
// FC612. Перевірка та розбір запису фізичного порту PROFINET 16#802A. Перевіряє заголовок, довжину й номер підслота; враховує змінну довжину назв і вирівнювання. TRUE означає достовірний стан фізичного зʼєднання. Блокування передавання кадрів менеджером MRP не є обривом фізичного зʼєднання.
   VAR_INPUT
      Length : UInt;   // Кількість байтів, фактично повернутих RDREC. Перевіряється перед доступом до буфера.
      ExpectedSubslot : UInt;   // Очікуваний підслот фізичного порту, наприклад 16#8001 для порту 1.
   END_VAR
   VAR_OUTPUT
      LinkUp : Bool;   // Фізичне зʼєднання встановлено. Використовувати лише за достовірного результату функції.
      LinkDown : Bool;   // Підтверджений стан відсутності фізичного зʼєднання. Не є доказом пошкодження саме кабелю.
      PortState : Byte;   // Стан передавання/блокування порту з отриманого запису; окремий від фізичного LinkState.
      LinkState : Byte;   // Стан фізичного зʼєднання з отриманого запису. Значення з невизначеним станом не приймаються.
   END_VAR
   VAR_IN_OUT
      Data : Array[0..1023] of Byte;   // Буфер прочитаного запису. Функція читає дані та не змінює їх.
   END_VAR
   VAR_TEMP
      n : DInt;   // Перевірена робоча довжина запису в байтах.
      p : DInt;   // Поточна позиція розбору в буфері; перевіряється перед читанням полів.
      count : Int;   // Кількість сусідів, вказана в записі фізичного порту.
      i : Int;   // Індекс циклу обробки елементів.
   END_VAR
BEGIN
   // FC612. Перевірка та розбір запису фізичного порту PROFINET 16#802A. Перевіряє заголовок, довжину й номер підслота; враховує змінну довжину назв і вирівнювання. TRUE означає достовірний стан фізичного зʼєднання. Блокування передавання кадрів менеджером MRP не є обривом фізичного зʼєднання.
   // Функція лише розбирає вже прочитаний буфер; RDREC виконує FB615.
   // Початковий результат — недостовірний. RETURN припиняє розбір некоректного запису.
   // LinkUp і LinkDown можна використовувати лише разом із TRUE результату функції.

       #FC_MRP_DecodePort := FALSE;
       #LinkUp := FALSE;
       #LinkDown := FALSE;
       #PortState := 0;
       #LinkState := 0;
       #n := UINT_TO_DINT(#Length);
       IF (#n < 36) OR (#n > 1024) THEN RETURN; END_IF;
       // Очікується PDPortDataReal 16#020F версії 1.0; повна довжина запису включає заголовок.
       IF (#Data[0] <> 16#02) OR (#Data[1] <> 16#0F) OR
          (#Data[4] <> 1) OR (#Data[5] <> 0) THEN RETURN; END_IF;
       IF BYTE_TO_DINT(#Data[2]) * 256 + BYTE_TO_DINT(#Data[3]) + 4 <> #n THEN RETURN; END_IF;
       IF BYTE_TO_UINT(#Data[10]) * UINT#256 + BYTE_TO_UINT(#Data[11]) <> #ExpectedSubslot THEN RETURN; END_IF;
       // Пройти назви власного порту й сусідів змінної довжини; фіксовані зміщення тут непридатні.
       #p := 13 + BYTE_TO_DINT(#Data[12]);
       IF #p >= #n THEN RETURN; END_IF;
       #count := BYTE_TO_INT(#Data[#p]);
       #p := ((#p + 1 + 3) / 4) * 4;
       FOR #i := 1 TO #count DO
           IF #p >= #n THEN RETURN; END_IF;
           #p := #p + 1 + BYTE_TO_DINT(#Data[#p]);
           IF #p >= #n THEN RETURN; END_IF;
           #p := #p + 1 + BYTE_TO_DINT(#Data[#p]);
           #p := ((#p + 3) / 4) * 4;
           // Затримка лінії — 4 байти, MAC сусіда — 6 байтів, вирівнювання — 2 байти.
           #p := #p + 12;
           IF #p > #n THEN RETURN; END_IF;
       END_FOR;
       IF #p + 20 <> #n THEN RETURN; END_IF;
       #PortState := #Data[#p + 12];
       #LinkState := #Data[#p + 13];
       // Блокування передавання на порту є нормальним для менеджера MRP. Саме стан фізичного звʼязку
       // визначає Link Down; стани тестування, невідомий або неактивний не вважаються підтвердженим обривом.
       #LinkUp := #LinkState = 1;
       #LinkDown := (#LinkState = 2) OR (#LinkState = 6) OR (#LinkState = 7);
       #FC_MRP_DecodePort := #LinkUp OR #LinkDown;
END_FUNCTION

FUNCTION "FC_MRP_DecodeRing" : Bool   // FC613, SCL
{ S7_Optimized_Access := 'TRUE' }
VERSION : 1.0
// FC613. Перевірка та розбір запису стану MRP 16#8050 від менеджера кільця. Підтримує реалізовані формати 1.0/1.1/1.2 для одного домену. TRUE означає знайдений та перевірений стан кільця. Непідтримуваний формат, роль клієнта або пошкоджений запис дають FALSE.
   VAR_INPUT
      Length : UInt;   // Кількість байтів, фактично повернутих RDREC. Перевіряється перед доступом до буфера.
   END_VAR
   VAR_OUTPUT
      Closed : Bool;   // TRUE — кільце замкнене; FALSE — розімкнене, але лише якщо результат функції TRUE.
      Role : UInt;   // Роль MRP з отриманого запису. Значення 2 відповідає менеджеру кільця.
   END_VAR
   VAR_IN_OUT
      Data : Array[0..1023] of Byte;   // Буфер прочитаного запису. Функція читає дані та не змінює їх.
   END_VAR
   VAR_TEMP
      n : DInt;   // Перевірена робоча довжина запису в байтах.
      p : DInt;   // Поточна позиція розбору в буфері; перевіряється перед читанням полів.
      instanceBase : DInt;   // Початкова позиція структури домену MRP у буфері.
      blockEnd : DInt;   // Кінець поточного контейнера запису; вихід за цю межу заборонено.
      nextBlock : DInt;   // Обчислена позиція наступного вкладеного блока після перевірки довжини.
      blockType : UInt;   // Тип вкладеного блока запису MRP.
      state : UInt;   // Значення стану кільця: 0 — розімкнене, 1 — замкнене.
      minorVersion : Byte;   // Молодша версія формату запису MRP.
      found : Bool;   // Блок стану кільця вже знайдено; повторний блок відхиляється як неоднозначний.
   END_VAR
BEGIN
   // FC613. Перевірка та розбір запису стану MRP 16#8050 від менеджера кільця. Підтримує реалізовані формати 1.0/1.1/1.2 для одного домену. TRUE означає знайдений та перевірений стан кільця. Непідтримуваний формат, роль клієнта або пошкоджений запис дають FALSE.
   // Функція лише розбирає вже прочитаний буфер; RDREC виконує FB615.
   // Стан кільця приймається лише від менеджера; наявність пристроїв не доводить замкненість кільця.
   // Closed має значення лише тоді, коли результат функції TRUE.

       #FC_MRP_DecodeRing := FALSE;
       #Closed := FALSE;
       #Role := 0;
       #found := FALSE;
       #n := UINT_TO_DINT(#Length);
       IF (#n < 32) OR (#n > 1024) THEN RETURN; END_IF;
       IF (#Data[0] <> 16#02) OR (#Data[1] <> 16#12) OR (#Data[4] <> 1) THEN RETURN; END_IF;
       IF BYTE_TO_DINT(#Data[2]) * 256 + BYTE_TO_DINT(#Data[3]) + 4 <> #n THEN RETURN; END_IF;
       #minorVersion := #Data[5];
       #instanceBase := 0;
       #blockEnd := #n;
       IF #minorVersion = 2 THEN
           // У цій конфігурації один домен MRP. Багатодоменний запис відхиляється, щоб уникнути неоднозначності.
           IF (#Data[7] <> 1) OR (#n < 40) THEN RETURN; END_IF;
           #instanceBase := 8;
           IF (#Data[8] <> 16#02) OR (#Data[9] <> 16#32) OR
              (#Data[12] <> 1) OR (#Data[13] <> 0) OR (#Data[15] <> 0) THEN RETURN; END_IF;
           #blockEnd := #instanceBase + BYTE_TO_DINT(#Data[10]) * 256 + BYTE_TO_DINT(#Data[11]) + 4;
           IF #blockEnd <> #n THEN RETURN; END_IF;
       ELSIF (#minorVersion <> 0) AND (#minorVersion <> 1) THEN
           RETURN;
       END_IF;
       #Role := BYTE_TO_UINT(#Data[#instanceBase + 24]) * UINT#256 + BYTE_TO_UINT(#Data[#instanceBase + 25]);
       // Стан кільця приймається лише тоді, коли адресований пристрій має роль менеджера MRP.
       IF #Role <> 2 THEN RETURN; END_IF;
       IF #minorVersion = 0 THEN
           #p := #instanceBase + 27 + BYTE_TO_DINT(#Data[#instanceBase + 26]) + 2;
       ELSE
           #p := #instanceBase + 29 + BYTE_TO_DINT(#Data[#instanceBase + 28]);
       END_IF;
       #p := ((#p + 3) / 4) * 4;
       IF #p > #blockEnd THEN RETURN; END_IF;
       WHILE #p + 6 <= #blockEnd DO
           #blockType := BYTE_TO_UINT(#Data[#p]) * UINT#256 + BYTE_TO_UINT(#Data[#p + 1]);
           #nextBlock := #p + BYTE_TO_DINT(#Data[#p + 2]) * 256 + BYTE_TO_DINT(#Data[#p + 3]) + 4;
           IF (#nextBlock < #p + 6) OR (#nextBlock > #blockEnd) THEN RETURN; END_IF;
           IF #blockType = UINT#16#0219 THEN
               IF #found OR (#nextBlock <> #p + 8) OR
                  (#Data[#p + 4] <> 1) OR (#Data[#p + 5] <> 0) THEN RETURN; END_IF;
               #state := BYTE_TO_UINT(#Data[#p + 6]) * UINT#256 + BYTE_TO_UINT(#Data[#p + 7]);
               IF #state > 1 THEN RETURN; END_IF;
               #Closed := #state = 1;
               #found := TRUE;
           END_IF;
           #p := #nextBlock;
       END_WHILE;
       #FC_MRP_DecodeRing := #found AND (#p = #blockEnd);
END_FUNCTION

FUNCTION "FC_MRP_Publish" : Void   // FC614, SCL
{ S7_Optimized_Access := 'TRUE' }
VERSION : 1.0
// FC614. Циклічна точка входу діагностики кільця. Спочатку викликає DB_Diag_Prof з ідентифікатором системи PROFINET IO, потім переносить чотири підтверджені ознаки Link Down у наявні теги червоних хрестиків HMI. Викликається з мережі 25 FC_Diagnostic.
BEGIN
   // FC614. Циклічна точка входу діагностики кільця. Спочатку викликає DB_Diag_Prof з ідентифікатором системи PROFINET IO, потім переносить чотири підтверджені ознаки Link Down у наявні теги червоних хрестиків HMI. Викликається з мережі 25 FC_Diagnostic.
   // Порядок важливий: спочатку оновити діагностику, потім передати результати на HMI.
   // Назви наявних тегів зі словом SCALAMCE збережено для сумісності з HMI.
   // Недоступність станції сама по собі не задає хрестик обриву; потрібні достовірні дані фізичного порту.

       "DB_Diag_Prof"(IO_System := "Local~PROFINET_IO-System");
       "HMI_DB".Diagnostics.Ring_PLC_HMI_NOK := "DB_Diag_Prof".Segment_PLC_HMI_Down;
       "HMI_DB".Diagnostics.Ring_PLC_SCALAMCE_NOK := "DB_Diag_Prof".Segment_PLC_SCALANCE_Down;
       "HMI_DB".Diagnostics.Ring_SCALAMCE_CU_NOK := "DB_Diag_Prof".Segment_SCALANCE_CU_Down;
       "HMI_DB".Diagnostics.Ring_HMI_CU_NOK := "DB_Diag_Prof".Segment_HMI_CU_Down;
END_FUNCTION

// folder: 700_Calibration

FUNCTION "FC_CalibrationCall" : Void   // FC700, LAD
TITLE = Калібровка енкодерів механізмів крана
{ S7_Optimized_Access := 'TRUE' }
VERSION : 0.1
   VAR_TEMP
      TempRemainingSeconds : UDInt;
   END_VAR
   VAR_TEMP   // added for the SCL form of the ladder/FBD networks
      _w1 : Bool;
   END_VAR
BEGIN

REGION Network 1: Калібровка механізму підйома
END_REGION

REGION Network 2 (SCL): Формування цільової координати у мм для пресету енкодера
   "DB_Calibration".Hoist.PresetTargetPosition_mm :=
   "DB_Calibration".Hoist.ReferencePosition_mm
   + "DB_Calibration".Hoist.VirtualOffset_mm
   + "DB_Calibration".Hoist.TravelAfterReference_mm;
END_REGION

REGION Network 3: Підготовка значення в інкрементах для пресету енкодера
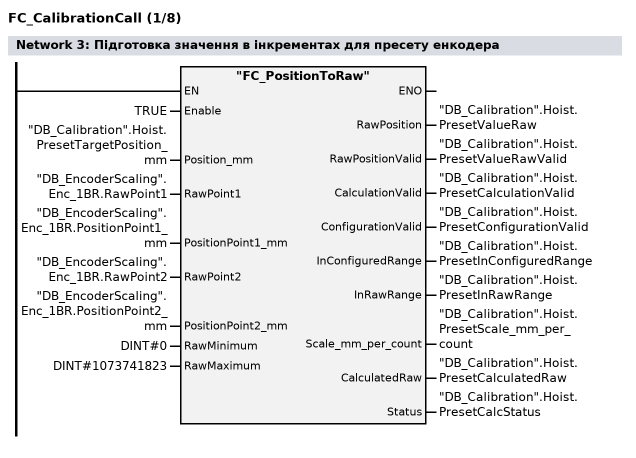
   RUNG wire#powerrail
      "FC_PositionToRaw"(Enable := TRUE, Position_mm := "DB_Calibration".Hoist.PresetTargetPosition_mm, RawPoint1 := "DB_EncoderScaling".Enc_1BR.RawPoint1, PositionPoint1_mm := "DB_EncoderScaling".Enc_1BR.PositionPoint1_mm, RawPoint2 := "DB_EncoderScaling".Enc_1BR.RawPoint2, PositionPoint2_mm := "DB_EncoderScaling".Enc_1BR.PositionPoint2_mm, RawMinimum := DINT#0, RawMaximum := DINT#1073741823, RawPosition => "DB_Calibration".Hoist.PresetValueRaw, RawPositionValid => "DB_Calibration".Hoist.PresetValueRawValid, CalculationValid => "DB_Calibration".Hoist.PresetCalculationValid, ConfigurationValid => "DB_Calibration".Hoist.PresetConfigurationValid, InConfiguredRange => "DB_Calibration".Hoist.PresetInConfiguredRange, InRawRange => "DB_Calibration".Hoist.PresetInRawRange, Scale_mm_per_count => "DB_Calibration".Hoist.PresetScale_mm_per_count, CalculatedRaw => "DB_Calibration".Hoist.PresetCalculatedRaw, Status => "DB_Calibration".Hoist.PresetCalcStatus)
   END_RUNG
   // the same network as SCL:
   "FC_PositionToRaw"(Enable := TRUE,
                      Position_mm := "DB_Calibration".Hoist.PresetTargetPosition_mm,
                      RawPoint1 := "DB_EncoderScaling".Enc_1BR.RawPoint1,
                      PositionPoint1_mm := "DB_EncoderScaling".Enc_1BR.PositionPoint1_mm,
                      RawPoint2 := "DB_EncoderScaling".Enc_1BR.RawPoint2,
                      PositionPoint2_mm := "DB_EncoderScaling".Enc_1BR.PositionPoint2_mm,
                      RawMinimum := DINT#0,
                      RawMaximum := DINT#1073741823,
                      RawPosition => "DB_Calibration".Hoist.PresetValueRaw,
                      RawPositionValid => "DB_Calibration".Hoist.PresetValueRawValid,
                      CalculationValid => "DB_Calibration".Hoist.PresetCalculationValid,
                      ConfigurationValid => "DB_Calibration".Hoist.PresetConfigurationValid,
                      InConfiguredRange => "DB_Calibration".Hoist.PresetInConfiguredRange,
                      InRawRange => "DB_Calibration".Hoist.PresetInRawRange,
                      Scale_mm_per_count => "DB_Calibration".Hoist.PresetScale_mm_per_count,
                      CalculatedRaw => "DB_Calibration".Hoist.PresetCalculatedRaw,
                      Status => "DB_Calibration".Hoist.PresetCalcStatus);
END_REGION

REGION Network 4: Калібровка енкодера енкодера 1BR механізму підйома
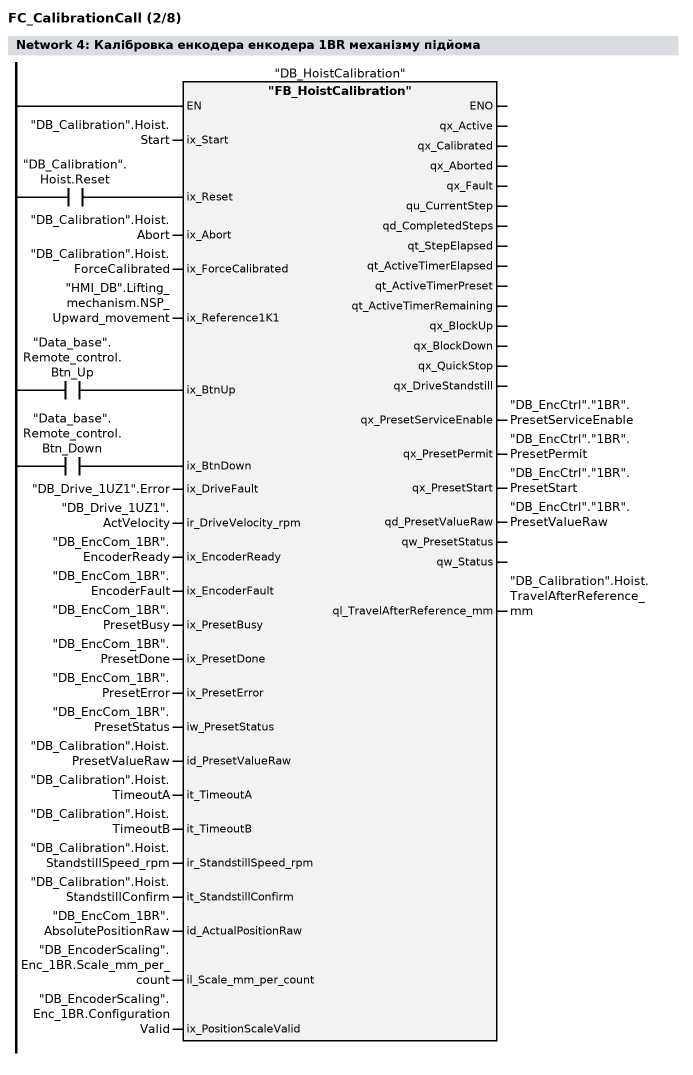
   RUNG wire#powerrail
      "DB_HoistCalibration"(ix_Reset := wire#w1, ix_BtnUp := wire#w2, ix_BtnDown := wire#w3, ix_Start := "DB_Calibration".Hoist.Start, ix_Abort := "DB_Calibration".Hoist.Abort, ix_ForceCalibrated := "DB_Calibration".Hoist.ForceCalibrated, ix_Reference1K1 := "HMI_DB".Lifting_mechanism.NSP_Upward_movement, ix_DriveFault := "DB_Drive_1UZ1".Error, ir_DriveVelocity_rpm := "DB_Drive_1UZ1".ActVelocity, ix_EncoderReady := "DB_EncCom_1BR".EncoderReady, ix_EncoderFault := "DB_EncCom_1BR".EncoderFault, ix_PresetBusy := "DB_EncCom_1BR".PresetBusy, ix_PresetDone := "DB_EncCom_1BR".PresetDone, ix_PresetError := "DB_EncCom_1BR".PresetError, iw_PresetStatus := "DB_EncCom_1BR".PresetStatus, id_PresetValueRaw := "DB_Calibration".Hoist.PresetValueRaw, it_TimeoutA := "DB_Calibration".Hoist.TimeoutA, it_TimeoutB := "DB_Calibration".Hoist.TimeoutB, ir_StandstillSpeed_rpm := "DB_Calibration".Hoist.StandstillSpeed_rpm, it_StandstillConfirm := "DB_Calibration".Hoist.StandstillConfirm, id_ActualPositionRaw := "DB_EncCom_1BR".AbsolutePositionRaw, il_Scale_mm_per_count := "DB_EncoderScaling".Enc_1BR.Scale_mm_per_count, ix_PositionScaleValid := "DB_EncoderScaling".Enc_1BR.ConfigurationValid, qx_Active =>, qx_Calibrated =>, qx_Aborted =>, qx_Fault =>, qu_CurrentStep =>, qd_CompletedSteps =>, qt_StepElapsed =>, qt_ActiveTimerElapsed =>, qt_ActiveTimerPreset =>, qt_ActiveTimerRemaining =>, qx_BlockUp =>, qx_BlockDown =>, qx_QuickStop =>, qx_DriveStandstill =>, qx_PresetServiceEnable => "DB_EncCtrl"."1BR".PresetServiceEnable, qx_PresetPermit => "DB_EncCtrl"."1BR".PresetPermit, qx_PresetStart => "DB_EncCtrl"."1BR".PresetStart, qd_PresetValueRaw => "DB_EncCtrl"."1BR".PresetValueRaw, qw_PresetStatus =>, qw_Status =>, ql_TravelAfterReference_mm => "DB_Calibration".Hoist.TravelAfterReference_mm)
   END_RUNG
   RUNG wire#powerrail
      Contact( "DB_Calibration".Hoist.Reset )
   END_RUNG wire#w1
   RUNG wire#powerrail
      Contact( "Data_base".Remote_control.Btn_Up )
   END_RUNG wire#w2
   RUNG wire#powerrail
      Contact( "Data_base".Remote_control.Btn_Down )
   END_RUNG wire#w3
   // the same network as SCL:
   "DB_HoistCalibration"(ix_Start := "DB_Calibration".Hoist.Start,   // "FB_HoistCalibration"
                         ix_Reset := "DB_Calibration".Hoist.Reset,
                         ix_Abort := "DB_Calibration".Hoist.Abort,
                         ix_ForceCalibrated := "DB_Calibration".Hoist.ForceCalibrated,
                         ix_Reference1K1 := "HMI_DB".Lifting_mechanism.NSP_Upward_movement,
                         ix_BtnUp := "Data_base".Remote_control.Btn_Up,
                         ix_BtnDown := "Data_base".Remote_control.Btn_Down,
                         ix_DriveFault := "DB_Drive_1UZ1".Error,
                         ir_DriveVelocity_rpm := "DB_Drive_1UZ1".ActVelocity,
                         ix_EncoderReady := "DB_EncCom_1BR".EncoderReady,
                         ix_EncoderFault := "DB_EncCom_1BR".EncoderFault,
                         ix_PresetBusy := "DB_EncCom_1BR".PresetBusy,
                         ix_PresetDone := "DB_EncCom_1BR".PresetDone,
                         ix_PresetError := "DB_EncCom_1BR".PresetError,
                         iw_PresetStatus := "DB_EncCom_1BR".PresetStatus,
                         id_PresetValueRaw := "DB_Calibration".Hoist.PresetValueRaw,
                         it_TimeoutA := "DB_Calibration".Hoist.TimeoutA,
                         it_TimeoutB := "DB_Calibration".Hoist.TimeoutB,
                         ir_StandstillSpeed_rpm := "DB_Calibration".Hoist.StandstillSpeed_rpm,
                         it_StandstillConfirm := "DB_Calibration".Hoist.StandstillConfirm,
                         id_ActualPositionRaw := "DB_EncCom_1BR".AbsolutePositionRaw,
                         il_Scale_mm_per_count := "DB_EncoderScaling".Enc_1BR.Scale_mm_per_count,
                         ix_PositionScaleValid := "DB_EncoderScaling".Enc_1BR.ConfigurationValid,
                         qx_PresetServiceEnable => "DB_EncCtrl"."1BR".PresetServiceEnable,
                         qx_PresetPermit => "DB_EncCtrl"."1BR".PresetPermit,
                         qx_PresetStart => "DB_EncCtrl"."1BR".PresetStart,
                         qd_PresetValueRaw => "DB_EncCtrl"."1BR".PresetValueRaw,
                         ql_TravelAfterReference_mm => "DB_Calibration".Hoist.TravelAfterReference_mm);
END_REGION

REGION Network 5: Діагностика калібровки енкодера 1BR механізму підйома
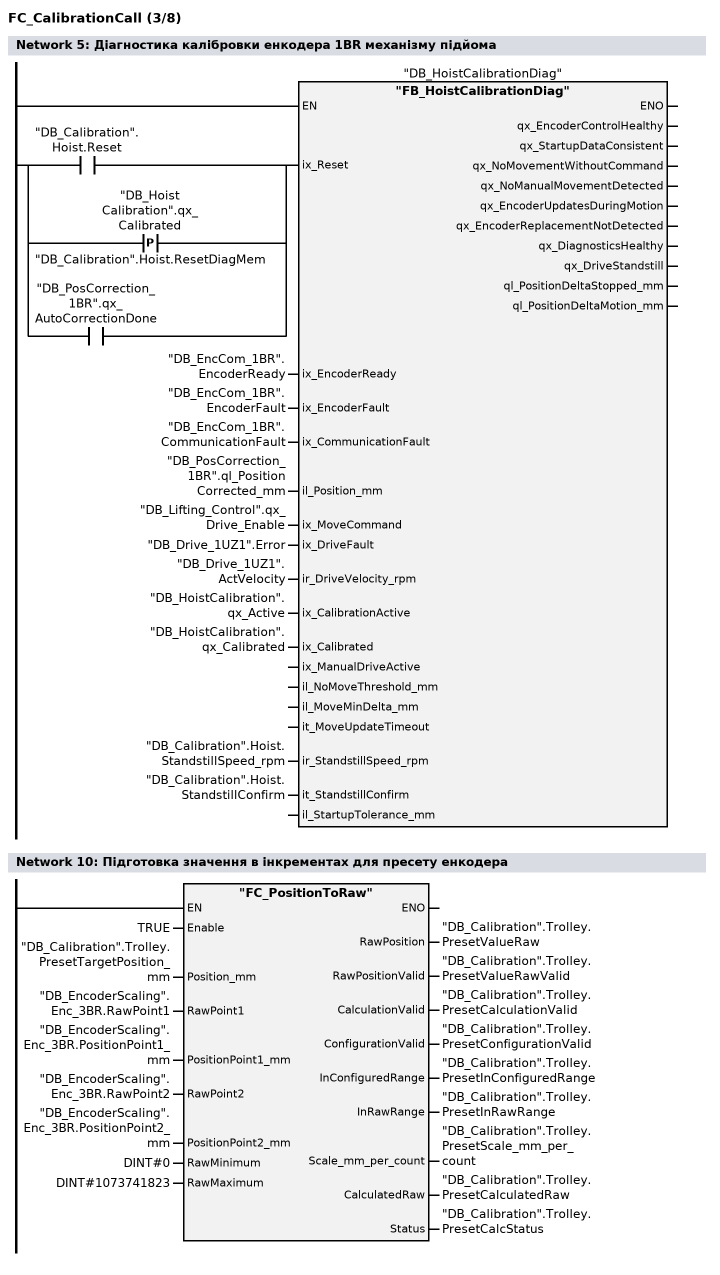
   RUNG wire#powerrail
      "DB_HoistCalibrationDiag"(ix_Reset := wire#w1, ix_EncoderReady := "DB_EncCom_1BR".EncoderReady, ix_EncoderFault := "DB_EncCom_1BR".EncoderFault, ix_CommunicationFault := "DB_EncCom_1BR".CommunicationFault, il_Position_mm := "DB_PosCorrection_1BR".ql_PositionCorrected_mm, ix_MoveCommand := "DB_Lifting_Control".qx_Drive_Enable, ix_DriveFault := "DB_Drive_1UZ1".Error, ir_DriveVelocity_rpm := "DB_Drive_1UZ1".ActVelocity, ix_CalibrationActive := "DB_HoistCalibration".qx_Active, ix_Calibrated := "DB_HoistCalibration".qx_Calibrated, ix_ManualDriveActive :=, il_NoMoveThreshold_mm :=, il_MoveMinDelta_mm :=, it_MoveUpdateTimeout :=, ir_StandstillSpeed_rpm := "DB_Calibration".Hoist.StandstillSpeed_rpm, it_StandstillConfirm := "DB_Calibration".Hoist.StandstillConfirm, il_StartupTolerance_mm :=, qx_EncoderControlHealthy =>, qx_StartupDataConsistent =>, qx_NoMovementWithoutCommand =>, qx_NoManualMovementDetected =>, qx_EncoderUpdatesDuringMotion =>, qx_EncoderReplacementNotDetected =>, qx_DiagnosticsHealthy =>, qx_DriveStandstill =>, ql_PositionDeltaStopped_mm =>, ql_PositionDeltaMotion_mm =>)
   END_RUNG
   RUNG wire#powerrail
      Contact( "DB_Calibration".Hoist.Reset )
   END_RUNG wire#w1
   RUNG wire#powerrail
      P_Contact(operand := "DB_HoistCalibration".qx_Calibrated, bit := "DB_Calibration".Hoist.ResetDiagMem)
   END_RUNG wire#w1
   RUNG wire#powerrail
      Contact( "DB_PosCorrection_1BR".qx_AutoCorrectionDone )
   END_RUNG wire#w1
   // the same network as SCL:
   #_w1 := "DB_HoistCalibration".qx_Calibrated AND NOT "DB_Calibration".Hoist.ResetDiagMem;   // rising edge of "DB_HoistCalibration".qx_Calibrated
   "DB_Calibration".Hoist.ResetDiagMem := "DB_HoistCalibration".qx_Calibrated;
   "DB_HoistCalibrationDiag"(ix_Reset := "DB_Calibration".Hoist.Reset OR #_w1 OR "DB_PosCorrection_1BR".qx_AutoCorrectionDone,   // "FB_HoistCalibrationDiag"
                           ix_EncoderReady := "DB_EncCom_1BR".EncoderReady,
                           ix_EncoderFault := "DB_EncCom_1BR".EncoderFault,
                           ix_CommunicationFault := "DB_EncCom_1BR".CommunicationFault,
                           il_Position_mm := "DB_PosCorrection_1BR".ql_PositionCorrected_mm,
                           ix_MoveCommand := "DB_Lifting_Control".qx_Drive_Enable,
                           ix_DriveFault := "DB_Drive_1UZ1".Error,
                           ir_DriveVelocity_rpm := "DB_Drive_1UZ1".ActVelocity,
                           ix_CalibrationActive := "DB_HoistCalibration".qx_Active,
                           ix_Calibrated := "DB_HoistCalibration".qx_Calibrated,
                           ir_StandstillSpeed_rpm := "DB_Calibration".Hoist.StandstillSpeed_rpm,
                           it_StandstillConfirm := "DB_Calibration".Hoist.StandstillConfirm);
END_REGION

REGION Network 6 (SCL): Калібровка підйома - дані на візуалізацію
   // Основний стан процедури калібровки
   "HMI_DB".Calibration.Hoist.Active :=
   "DB_HoistCalibration".qx_Active;

   "HMI_DB".Calibration.Hoist.Calibrated :=
   "DB_HoistCalibration".qx_Calibrated;

   "HMI_DB".Calibration.Hoist.Fault :=
   "DB_HoistCalibration".qx_Fault;

   "HMI_DB".Calibration.Hoist.Aborted :=
   "DB_HoistCalibration".qx_Aborted;


   // Поточний крок та завершені кроки
   "HMI_DB".Calibration.Hoist.CurrentStep :=
   "DB_HoistCalibration".qu_CurrentStep;

   "HMI_DB".Calibration.Hoist.CompletedSteps :=
   "DB_HoistCalibration".qd_CompletedSteps;


   // Реперний кінцевик 1K1
   // Беремо той самий сигнал, який бачить FB_HoistCalibration
   "HMI_DB".Calibration.Hoist.Reference1K1 :=
   "DB_HoistCalibration".ix_Reference1K1;


   // Поточне положення механізму
   "HMI_DB".Calibration.Hoist.Position_mm :=
   "DB_PosCorrection_1BR".qd_PositionCorrectedRounded_mm;


   // Фактична швидкість привода
   // Беремо те саме значення, яке використовує сіквенсер калібровки
   "HMI_DB".Calibration.Hoist.DriveVelocity_rpm :=
   "DB_HoistCalibration".ir_DriveVelocity_rpm;


   // Залишок часу активного таймера
   "HMI_DB".Calibration.Hoist.TimerRemaining :=
   "DB_HoistCalibration".qt_ActiveTimerRemaining;

   // Перетворюємо час у форматі TIME на загальну кількість секунд
   #TempRemainingSeconds :=
   TIME_TO_UDINT("DB_HoistCalibration".qt_ActiveTimerRemaining) / UDINT#1000;

   // Повні хвилини
   "HMI_DB".Calibration.Hoist.TimerRemaining_Min :=
   UDINT_TO_UINT(#TempRemainingSeconds / UDINT#60);

   // Залишок секунд
   "HMI_DB".Calibration.Hoist.TimerRemaining_Sec :=
   UDINT_TO_UINT(#TempRemainingSeconds MOD UDINT#60);


   // ============================================================
   // HMI mapping - completed calibration steps
   // ============================================================

   "HMI_DB".Calibration.Hoist.Steps_Completed.Step10 :=
   "DB_HoistCalibration".qd_CompletedSteps.%X0;

   "HMI_DB".Calibration.Hoist.Steps_Completed.Step20 :=
   "DB_HoistCalibration".qd_CompletedSteps.%X1;

   "HMI_DB".Calibration.Hoist.Steps_Completed.Step30 :=
   "DB_HoistCalibration".qd_CompletedSteps.%X2;

   "HMI_DB".Calibration.Hoist.Steps_Completed.Step40 :=
   "DB_HoistCalibration".qd_CompletedSteps.%X3;

   "HMI_DB".Calibration.Hoist.Steps_Completed.Step50 :=
   "DB_HoistCalibration".qd_CompletedSteps.%X4;

   "HMI_DB".Calibration.Hoist.Steps_Completed.Step60 :=
   "DB_HoistCalibration".qd_CompletedSteps.%X5;

   "HMI_DB".Calibration.Hoist.Steps_Completed.Step70 :=
   "DB_HoistCalibration".qd_CompletedSteps.%X6;

   "HMI_DB".Calibration.Hoist.Steps_Completed.Step80 :=
   "DB_HoistCalibration".qd_CompletedSteps.%X7;

   "HMI_DB".Calibration.Hoist.Steps_Completed.Step90 :=
   "DB_HoistCalibration".qd_CompletedSteps.%X8;

   "HMI_DB".Calibration.Hoist.Steps_Completed.Step100 :=
   "DB_HoistCalibration".qd_CompletedSteps.%X9;

   "HMI_DB".Calibration.Hoist.Steps_Completed.Step110 :=
   "DB_HoistCalibration".qd_CompletedSteps.%X10;

   "HMI_DB".Calibration.Hoist.Steps_Completed.Step120 :=
   "DB_HoistCalibration".qd_CompletedSteps.%X11;

   "HMI_DB".Calibration.Hoist.Steps_Completed.Step130 :=
   "DB_HoistCalibration".qd_CompletedSteps.%X12;

   // ============================================================
   // HMI mapping - active calibration steps
   // ============================================================

   "HMI_DB".Calibration.Hoist.Steps_Active.Step10 :=
   "HMI_DB".Calibration.Hoist.CurrentStep = UINT#10;

   "HMI_DB".Calibration.Hoist.Steps_Active.Step20 :=
   "HMI_DB".Calibration.Hoist.CurrentStep = UINT#20;

   "HMI_DB".Calibration.Hoist.Steps_Active.Step30 :=
   "HMI_DB".Calibration.Hoist.CurrentStep = UINT#30;

   "HMI_DB".Calibration.Hoist.Steps_Active.Step40 :=
   "HMI_DB".Calibration.Hoist.CurrentStep = UINT#40;

   "HMI_DB".Calibration.Hoist.Steps_Active.Step50 :=
   "HMI_DB".Calibration.Hoist.CurrentStep = UINT#50;

   "HMI_DB".Calibration.Hoist.Steps_Active.Step60 :=
   "HMI_DB".Calibration.Hoist.CurrentStep = UINT#60;

   "HMI_DB".Calibration.Hoist.Steps_Active.Step70 :=
   "HMI_DB".Calibration.Hoist.CurrentStep = UINT#70;

   "HMI_DB".Calibration.Hoist.Steps_Active.Step80 :=
   "HMI_DB".Calibration.Hoist.CurrentStep = UINT#80;

   "HMI_DB".Calibration.Hoist.Steps_Active.Step90 :=
   "HMI_DB".Calibration.Hoist.CurrentStep = UINT#90;

   "HMI_DB".Calibration.Hoist.Steps_Active.Step100 :=
   "HMI_DB".Calibration.Hoist.CurrentStep = UINT#100;

   "HMI_DB".Calibration.Hoist.Steps_Active.Step110 :=
   "HMI_DB".Calibration.Hoist.CurrentStep = UINT#110;

   "HMI_DB".Calibration.Hoist.Steps_Active.Step120 :=
   "HMI_DB".Calibration.Hoist.CurrentStep = UINT#120;

   "HMI_DB".Calibration.Hoist.Steps_Active.Step130 :=
   "HMI_DB".Calibration.Hoist.CurrentStep = UINT#130;

   // ============================================================
   // HMI mapping - hoist calibration diagnostics
   // ============================================================

   "HMI_DB".Calibration.Hoist.Diagnostics.EncoderControlHealthy :=
   "DB_HoistCalibrationDiag".qx_EncoderControlHealthy;

   "HMI_DB".Calibration.Hoist.Diagnostics.StartupDataConsistent :=
   "DB_HoistCalibrationDiag".qx_StartupDataConsistent;

   "HMI_DB".Calibration.Hoist.Diagnostics.NoMovementWithoutCommand :=
   "DB_HoistCalibrationDiag".qx_NoMovementWithoutCommand;

   "HMI_DB".Calibration.Hoist.Diagnostics.NoManualMovementDetected :=
   "DB_HoistCalibrationDiag".qx_NoManualMovementDetected;

   "HMI_DB".Calibration.Hoist.Diagnostics.EncoderUpdatesDuringMotion :=
   "DB_HoistCalibrationDiag".qx_EncoderUpdatesDuringMotion;

   "HMI_DB".Calibration.Hoist.Diagnostics.EncoderReplacementNotDetected :=
   "DB_HoistCalibrationDiag".qx_EncoderReplacementNotDetected;
END_REGION

REGION Network 8: Калібровка механізму візка
END_REGION

REGION Network 9 (SCL): Формування цільової координати у мм для пресету енкодера
   "DB_Calibration".Trolley.PresetTargetPosition_mm :=
   "DB_Calibration".Trolley.ReferencePosition_mm
   + "DB_Calibration".Trolley.VirtualOffset_mm
   + "DB_Calibration".Trolley.TravelAfterReference_mm;
END_REGION

REGION Network 10: Підготовка значення в інкрементах для пресету енкодера
   RUNG wire#powerrail
      "FC_PositionToRaw"(Enable := TRUE, Position_mm := "DB_Calibration".Trolley.PresetTargetPosition_mm, RawPoint1 := "DB_EncoderScaling".Enc_3BR.RawPoint1, PositionPoint1_mm := "DB_EncoderScaling".Enc_3BR.PositionPoint1_mm, RawPoint2 := "DB_EncoderScaling".Enc_3BR.RawPoint2, PositionPoint2_mm := "DB_EncoderScaling".Enc_3BR.PositionPoint2_mm, RawMinimum := DINT#0, RawMaximum := DINT#1073741823, RawPosition => "DB_Calibration".Trolley.PresetValueRaw, RawPositionValid => "DB_Calibration".Trolley.PresetValueRawValid, CalculationValid => "DB_Calibration".Trolley.PresetCalculationValid, ConfigurationValid => "DB_Calibration".Trolley.PresetConfigurationValid, InConfiguredRange => "DB_Calibration".Trolley.PresetInConfiguredRange, InRawRange => "DB_Calibration".Trolley.PresetInRawRange, Scale_mm_per_count => "DB_Calibration".Trolley.PresetScale_mm_per_count, CalculatedRaw => "DB_Calibration".Trolley.PresetCalculatedRaw, Status => "DB_Calibration".Trolley.PresetCalcStatus)
   END_RUNG
   // the same network as SCL:
   "FC_PositionToRaw"(Enable := TRUE,
                      Position_mm := "DB_Calibration".Trolley.PresetTargetPosition_mm,
                      RawPoint1 := "DB_EncoderScaling".Enc_3BR.RawPoint1,
                      PositionPoint1_mm := "DB_EncoderScaling".Enc_3BR.PositionPoint1_mm,
                      RawPoint2 := "DB_EncoderScaling".Enc_3BR.RawPoint2,
                      PositionPoint2_mm := "DB_EncoderScaling".Enc_3BR.PositionPoint2_mm,
                      RawMinimum := DINT#0,
                      RawMaximum := DINT#1073741823,
                      RawPosition => "DB_Calibration".Trolley.PresetValueRaw,
                      RawPositionValid => "DB_Calibration".Trolley.PresetValueRawValid,
                      CalculationValid => "DB_Calibration".Trolley.PresetCalculationValid,
                      ConfigurationValid => "DB_Calibration".Trolley.PresetConfigurationValid,
                      InConfiguredRange => "DB_Calibration".Trolley.PresetInConfiguredRange,
                      InRawRange => "DB_Calibration".Trolley.PresetInRawRange,
                      Scale_mm_per_count => "DB_Calibration".Trolley.PresetScale_mm_per_count,
                      CalculatedRaw => "DB_Calibration".Trolley.PresetCalculatedRaw,
                      Status => "DB_Calibration".Trolley.PresetCalcStatus);
END_REGION

REGION Network 11: Калібровка енкодера 3BR механізму візка
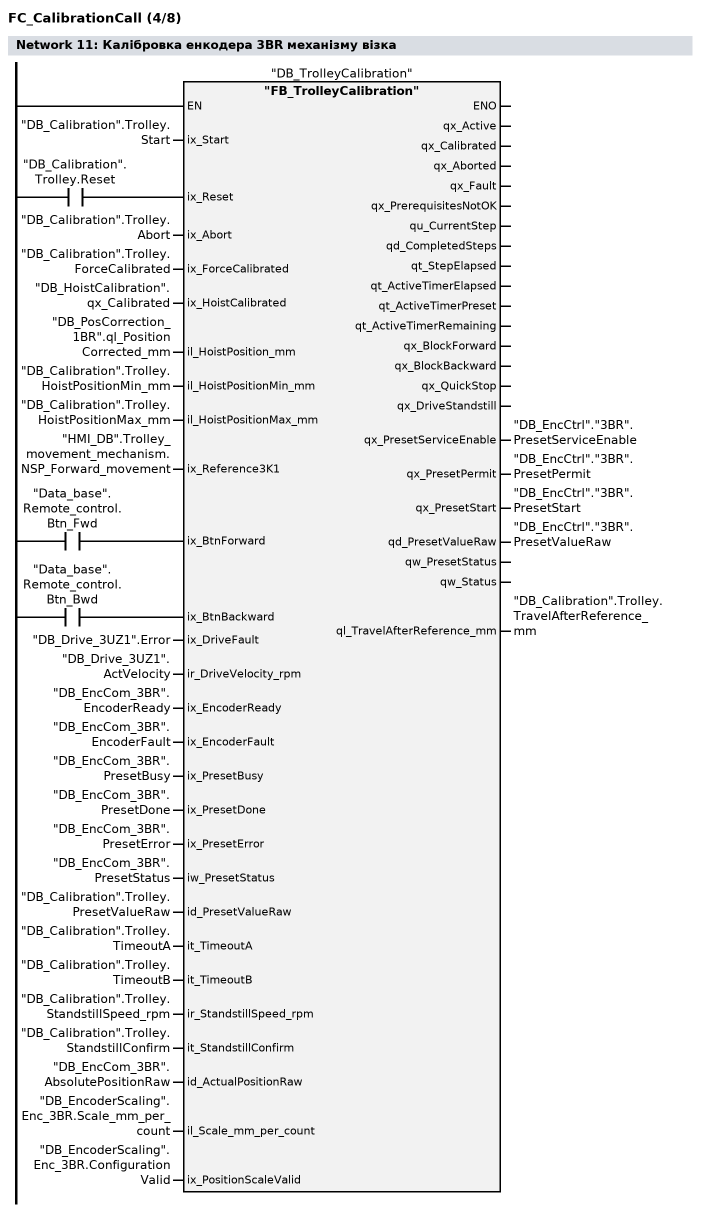
   RUNG wire#powerrail
      "DB_TrolleyCalibration"(ix_Reset := wire#w1, ix_BtnForward := wire#w2, ix_BtnBackward := wire#w3, ix_Start := "DB_Calibration".Trolley.Start, ix_Abort := "DB_Calibration".Trolley.Abort, ix_ForceCalibrated := "DB_Calibration".Trolley.ForceCalibrated, ix_HoistCalibrated := "DB_HoistCalibration".qx_Calibrated, il_HoistPosition_mm := "DB_PosCorrection_1BR".ql_PositionCorrected_mm, il_HoistPositionMin_mm := "DB_Calibration".Trolley.HoistPositionMin_mm, il_HoistPositionMax_mm := "DB_Calibration".Trolley.HoistPositionMax_mm, ix_Reference3K1 := "HMI_DB".Trolley_movement_mechanism.NSP_Forward_movement, ix_DriveFault := "DB_Drive_3UZ1".Error, ir_DriveVelocity_rpm := "DB_Drive_3UZ1".ActVelocity, ix_EncoderReady := "DB_EncCom_3BR".EncoderReady, ix_EncoderFault := "DB_EncCom_3BR".EncoderFault, ix_PresetBusy := "DB_EncCom_3BR".PresetBusy, ix_PresetDone := "DB_EncCom_3BR".PresetDone, ix_PresetError := "DB_EncCom_3BR".PresetError, iw_PresetStatus := "DB_EncCom_3BR".PresetStatus, id_PresetValueRaw := "DB_Calibration".Trolley.PresetValueRaw, it_TimeoutA := "DB_Calibration".Trolley.TimeoutA, it_TimeoutB := "DB_Calibration".Trolley.TimeoutB, ir_StandstillSpeed_rpm := "DB_Calibration".Trolley.StandstillSpeed_rpm, it_StandstillConfirm := "DB_Calibration".Trolley.StandstillConfirm, id_ActualPositionRaw := "DB_EncCom_3BR".AbsolutePositionRaw, il_Scale_mm_per_count := "DB_EncoderScaling".Enc_3BR.Scale_mm_per_count, ix_PositionScaleValid := "DB_EncoderScaling".Enc_3BR.ConfigurationValid, qx_Active =>, qx_Calibrated =>, qx_Aborted =>, qx_Fault =>, qx_PrerequisitesNotOK =>, qu_CurrentStep =>, qd_CompletedSteps =>, qt_StepElapsed =>, qt_ActiveTimerElapsed =>, qt_ActiveTimerPreset =>, qt_ActiveTimerRemaining =>, qx_BlockForward =>, qx_BlockBackward =>, qx_QuickStop =>, qx_DriveStandstill =>, qx_PresetServiceEnable => "DB_EncCtrl"."3BR".PresetServiceEnable, qx_PresetPermit => "DB_EncCtrl"."3BR".PresetPermit, qx_PresetStart => "DB_EncCtrl"."3BR".PresetStart, qd_PresetValueRaw => "DB_EncCtrl"."3BR".PresetValueRaw, qw_PresetStatus =>, qw_Status =>, ql_TravelAfterReference_mm => "DB_Calibration".Trolley.TravelAfterReference_mm)
   END_RUNG
   RUNG wire#powerrail
      Contact( "DB_Calibration".Trolley.Reset )
   END_RUNG wire#w1
   RUNG wire#powerrail
      Contact( "Data_base".Remote_control.Btn_Fwd )
   END_RUNG wire#w2
   RUNG wire#powerrail
      Contact( "Data_base".Remote_control.Btn_Bwd )
   END_RUNG wire#w3
   // the same network as SCL:
   "DB_TrolleyCalibration"(ix_Start := "DB_Calibration".Trolley.Start,   // "FB_TrolleyCalibration"
                           ix_Reset := "DB_Calibration".Trolley.Reset,
                           ix_Abort := "DB_Calibration".Trolley.Abort,
                           ix_ForceCalibrated := "DB_Calibration".Trolley.ForceCalibrated,
                           ix_HoistCalibrated := "DB_HoistCalibration".qx_Calibrated,
                           il_HoistPosition_mm := "DB_PosCorrection_1BR".ql_PositionCorrected_mm,
                           il_HoistPositionMin_mm := "DB_Calibration".Trolley.HoistPositionMin_mm,
                           il_HoistPositionMax_mm := "DB_Calibration".Trolley.HoistPositionMax_mm,
                           ix_Reference3K1 := "HMI_DB".Trolley_movement_mechanism.NSP_Forward_movement,
                           ix_BtnForward := "Data_base".Remote_control.Btn_Fwd,
                           ix_BtnBackward := "Data_base".Remote_control.Btn_Bwd,
                           ix_DriveFault := "DB_Drive_3UZ1".Error,
                           ir_DriveVelocity_rpm := "DB_Drive_3UZ1".ActVelocity,
                           ix_EncoderReady := "DB_EncCom_3BR".EncoderReady,
                           ix_EncoderFault := "DB_EncCom_3BR".EncoderFault,
                           ix_PresetBusy := "DB_EncCom_3BR".PresetBusy,
                           ix_PresetDone := "DB_EncCom_3BR".PresetDone,
                           ix_PresetError := "DB_EncCom_3BR".PresetError,
                           iw_PresetStatus := "DB_EncCom_3BR".PresetStatus,
                           id_PresetValueRaw := "DB_Calibration".Trolley.PresetValueRaw,
                           it_TimeoutA := "DB_Calibration".Trolley.TimeoutA,
                           it_TimeoutB := "DB_Calibration".Trolley.TimeoutB,
                           ir_StandstillSpeed_rpm := "DB_Calibration".Trolley.StandstillSpeed_rpm,
                           it_StandstillConfirm := "DB_Calibration".Trolley.StandstillConfirm,
                           id_ActualPositionRaw := "DB_EncCom_3BR".AbsolutePositionRaw,
                           il_Scale_mm_per_count := "DB_EncoderScaling".Enc_3BR.Scale_mm_per_count,
                           ix_PositionScaleValid := "DB_EncoderScaling".Enc_3BR.ConfigurationValid,
                           qx_PresetServiceEnable => "DB_EncCtrl"."3BR".PresetServiceEnable,
                           qx_PresetPermit => "DB_EncCtrl"."3BR".PresetPermit,
                           qx_PresetStart => "DB_EncCtrl"."3BR".PresetStart,
                           qd_PresetValueRaw => "DB_EncCtrl"."3BR".PresetValueRaw,
                           ql_TravelAfterReference_mm => "DB_Calibration".Trolley.TravelAfterReference_mm);
END_REGION

REGION Network 12: Діагностика калібровки енкодера 3BR механізму візка
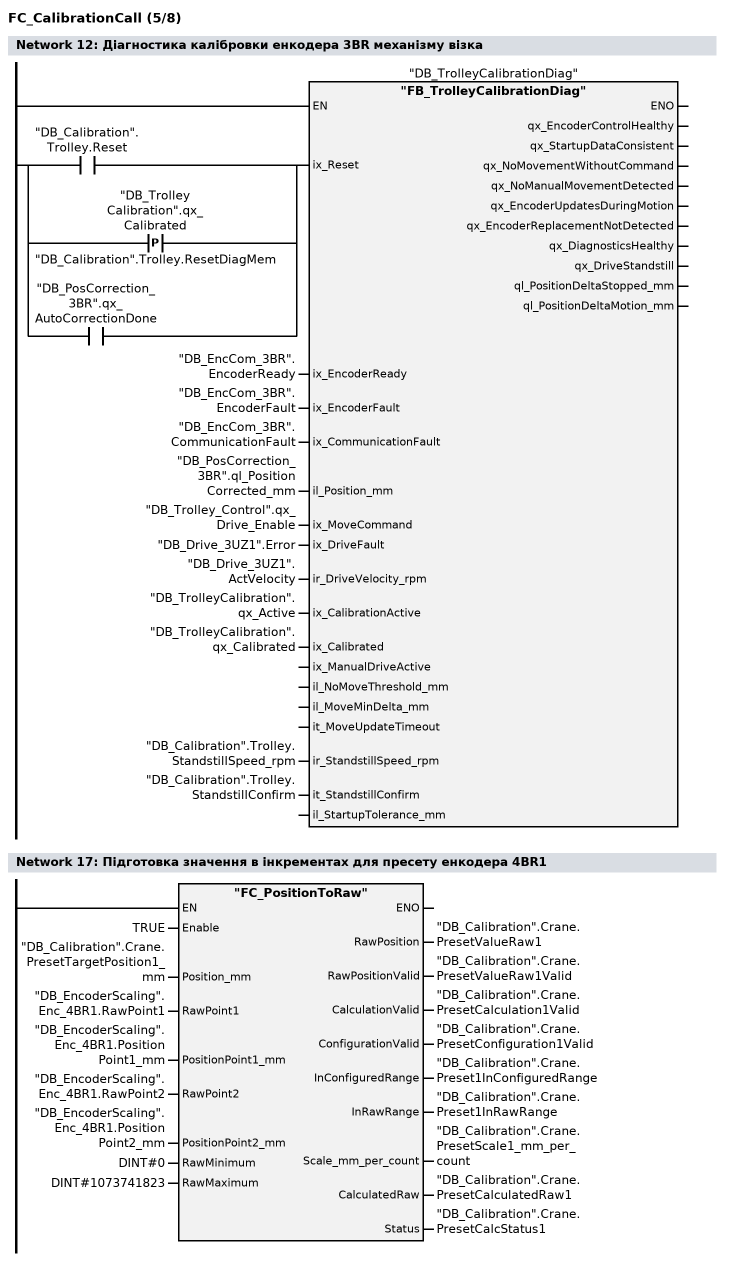
   RUNG wire#powerrail
      "DB_TrolleyCalibrationDiag"(ix_Reset := wire#w1, ix_EncoderReady := "DB_EncCom_3BR".EncoderReady, ix_EncoderFault := "DB_EncCom_3BR".EncoderFault, ix_CommunicationFault := "DB_EncCom_3BR".CommunicationFault, il_Position_mm := "DB_PosCorrection_3BR".ql_PositionCorrected_mm, ix_MoveCommand := "DB_Trolley_Control".qx_Drive_Enable, ix_DriveFault := "DB_Drive_3UZ1".Error, ir_DriveVelocity_rpm := "DB_Drive_3UZ1".ActVelocity, ix_CalibrationActive := "DB_TrolleyCalibration".qx_Active, ix_Calibrated := "DB_TrolleyCalibration".qx_Calibrated, ix_ManualDriveActive :=, il_NoMoveThreshold_mm :=, il_MoveMinDelta_mm :=, it_MoveUpdateTimeout :=, ir_StandstillSpeed_rpm := "DB_Calibration".Trolley.StandstillSpeed_rpm, it_StandstillConfirm := "DB_Calibration".Trolley.StandstillConfirm, il_StartupTolerance_mm :=, qx_EncoderControlHealthy =>, qx_StartupDataConsistent =>, qx_NoMovementWithoutCommand =>, qx_NoManualMovementDetected =>, qx_EncoderUpdatesDuringMotion =>, qx_EncoderReplacementNotDetected =>, qx_DiagnosticsHealthy =>, qx_DriveStandstill =>, ql_PositionDeltaStopped_mm =>, ql_PositionDeltaMotion_mm =>)
   END_RUNG
   RUNG wire#powerrail
      Contact( "DB_Calibration".Trolley.Reset )
   END_RUNG wire#w1
   RUNG wire#powerrail
      P_Contact(operand := "DB_TrolleyCalibration".qx_Calibrated, bit := "DB_Calibration".Trolley.ResetDiagMem)
   END_RUNG wire#w1
   RUNG wire#powerrail
      Contact( "DB_PosCorrection_3BR".qx_AutoCorrectionDone )
   END_RUNG wire#w1
   // the same network as SCL:
   #_w1 := "DB_TrolleyCalibration".qx_Calibrated AND NOT "DB_Calibration".Trolley.ResetDiagMem;   // rising edge of "DB_TrolleyCalibration".qx_Calibrated
   "DB_Calibration".Trolley.ResetDiagMem := "DB_TrolleyCalibration".qx_Calibrated;
   "DB_TrolleyCalibrationDiag"(ix_Reset := "DB_Calibration".Trolley.Reset OR #_w1 OR "DB_PosCorrection_3BR".qx_AutoCorrectionDone,   // "FB_TrolleyCalibrationDiag"
                           ix_EncoderReady := "DB_EncCom_3BR".EncoderReady,
                           ix_EncoderFault := "DB_EncCom_3BR".EncoderFault,
                           ix_CommunicationFault := "DB_EncCom_3BR".CommunicationFault,
                           il_Position_mm := "DB_PosCorrection_3BR".ql_PositionCorrected_mm,
                           ix_MoveCommand := "DB_Trolley_Control".qx_Drive_Enable,
                           ix_DriveFault := "DB_Drive_3UZ1".Error,
                           ir_DriveVelocity_rpm := "DB_Drive_3UZ1".ActVelocity,
                           ix_CalibrationActive := "DB_TrolleyCalibration".qx_Active,
                           ix_Calibrated := "DB_TrolleyCalibration".qx_Calibrated,
                           ir_StandstillSpeed_rpm := "DB_Calibration".Trolley.StandstillSpeed_rpm,
                           it_StandstillConfirm := "DB_Calibration".Trolley.StandstillConfirm);
END_REGION

REGION Network 13 (SCL): Калібровка візка - дані на візуалізацію
   // ============================================================
   // HMI mapping - trolley calibration
   // ============================================================

   "HMI_DB".Calibration.Trolley.Active :=
   "DB_TrolleyCalibration".qx_Active;

   "HMI_DB".Calibration.Trolley.Calibrated :=
   "DB_TrolleyCalibration".qx_Calibrated;

   "HMI_DB".Calibration.Trolley.Fault :=
   "DB_TrolleyCalibration".qx_Fault;

   "HMI_DB".Calibration.Trolley.Aborted :=
   "DB_TrolleyCalibration".qx_Aborted;

   "HMI_DB".Calibration.Trolley.PrerequisitesNotOK :=
   "DB_TrolleyCalibration".qx_PrerequisitesNotOK;

   "HMI_DB".Calibration.Trolley.CurrentStep :=
   "DB_TrolleyCalibration".qu_CurrentStep;

   "HMI_DB".Calibration.Trolley.CompletedSteps :=
   "DB_TrolleyCalibration".qd_CompletedSteps;


   // Current state of reference switch 3K1
   "HMI_DB".Calibration.Trolley.Reference3K1 :=
   "DB_TrolleyCalibration".ix_Reference3K1;


   // Current trolley position
   "HMI_DB".Calibration.Trolley.Position_mm :=
   "DB_PosCorrection_3BR".qd_PositionCorrectedRounded_mm;

   // Actual drive velocity
   // Use the same drive tag that is connected to
   // FB_TrolleyCalibration.ir_DriveVelocity_rpm
   "HMI_DB".Calibration.Trolley.DriveVelocity_rpm :=
   "DB_TrolleyCalibration".ir_DriveVelocity_rpm;

   // Active timer
   "HMI_DB".Calibration.Trolley.TimerRemaining :=
   "DB_TrolleyCalibration".qt_ActiveTimerRemaining;

   // ============================================================
   // HMI mapping - trolley calibration timer
   // ============================================================

   #TempRemainingSeconds :=
   TIME_TO_UDINT("DB_TrolleyCalibration".qt_ActiveTimerRemaining)
   / UDINT#1000;

   "HMI_DB".Calibration.Trolley.TimerRemaining_Min :=
   UDINT_TO_UINT(#TempRemainingSeconds / UDINT#60);

   "HMI_DB".Calibration.Trolley.TimerRemaining_Sec :=
   UDINT_TO_UINT(#TempRemainingSeconds MOD UDINT#60);

   // ============================================================
   // HMI mapping - trolley completed calibration steps
   // ============================================================

   "HMI_DB".Calibration.Trolley.Steps_Completed.Step10 :=
   "DB_TrolleyCalibration".qd_CompletedSteps.%X0;

   "HMI_DB".Calibration.Trolley.Steps_Completed.Step20 :=
   "DB_TrolleyCalibration".qd_CompletedSteps.%X1;

   "HMI_DB".Calibration.Trolley.Steps_Completed.Step30 :=
   "DB_TrolleyCalibration".qd_CompletedSteps.%X2;

   "HMI_DB".Calibration.Trolley.Steps_Completed.Step40 :=
   "DB_TrolleyCalibration".qd_CompletedSteps.%X3;

   "HMI_DB".Calibration.Trolley.Steps_Completed.Step50 :=
   "DB_TrolleyCalibration".qd_CompletedSteps.%X4;

   "HMI_DB".Calibration.Trolley.Steps_Completed.Step60 :=
   "DB_TrolleyCalibration".qd_CompletedSteps.%X5;

   "HMI_DB".Calibration.Trolley.Steps_Completed.Step70 :=
   "DB_TrolleyCalibration".qd_CompletedSteps.%X6;

   "HMI_DB".Calibration.Trolley.Steps_Completed.Step80 :=
   "DB_TrolleyCalibration".qd_CompletedSteps.%X7;

   "HMI_DB".Calibration.Trolley.Steps_Completed.Step90 :=
   "DB_TrolleyCalibration".qd_CompletedSteps.%X8;

   "HMI_DB".Calibration.Trolley.Steps_Completed.Step100 :=
   "DB_TrolleyCalibration".qd_CompletedSteps.%X9;

   "HMI_DB".Calibration.Trolley.Steps_Completed.Step110 :=
   "DB_TrolleyCalibration".qd_CompletedSteps.%X10;

   "HMI_DB".Calibration.Trolley.Steps_Completed.Step120 :=
   "DB_TrolleyCalibration".qd_CompletedSteps.%X11;

   "HMI_DB".Calibration.Trolley.Steps_Completed.Step130 :=
   "DB_TrolleyCalibration".qd_CompletedSteps.%X12;

   // ============================================================
   // HMI mapping - trolley active calibration steps
   // ============================================================

   "HMI_DB".Calibration.Trolley.Steps_Active.Step10 :=
   "HMI_DB".Calibration.Trolley.CurrentStep = UINT#10;

   "HMI_DB".Calibration.Trolley.Steps_Active.Step20 :=
   "HMI_DB".Calibration.Trolley.CurrentStep = UINT#20;

   "HMI_DB".Calibration.Trolley.Steps_Active.Step30 :=
   "HMI_DB".Calibration.Trolley.CurrentStep = UINT#30;

   "HMI_DB".Calibration.Trolley.Steps_Active.Step40 :=
   "HMI_DB".Calibration.Trolley.CurrentStep = UINT#40;

   "HMI_DB".Calibration.Trolley.Steps_Active.Step50 :=
   "HMI_DB".Calibration.Trolley.CurrentStep = UINT#50;

   "HMI_DB".Calibration.Trolley.Steps_Active.Step60 :=
   "HMI_DB".Calibration.Trolley.CurrentStep = UINT#60;

   "HMI_DB".Calibration.Trolley.Steps_Active.Step70 :=
   "HMI_DB".Calibration.Trolley.CurrentStep = UINT#70;

   "HMI_DB".Calibration.Trolley.Steps_Active.Step80 :=
   "HMI_DB".Calibration.Trolley.CurrentStep = UINT#80;

   "HMI_DB".Calibration.Trolley.Steps_Active.Step90 :=
   "HMI_DB".Calibration.Trolley.CurrentStep = UINT#90;

   "HMI_DB".Calibration.Trolley.Steps_Active.Step100 :=
   "HMI_DB".Calibration.Trolley.CurrentStep = UINT#100;

   "HMI_DB".Calibration.Trolley.Steps_Active.Step110 :=
   "HMI_DB".Calibration.Trolley.CurrentStep = UINT#110;

   "HMI_DB".Calibration.Trolley.Steps_Active.Step120 :=
   "HMI_DB".Calibration.Trolley.CurrentStep = UINT#120;

   "HMI_DB".Calibration.Trolley.Steps_Active.Step130 :=
   "HMI_DB".Calibration.Trolley.CurrentStep = UINT#130;


   // ============================================================
   // HMI mapping - trolley calibration diagnostics
   // ============================================================

   "HMI_DB".Calibration.Trolley.Diagnostics.EncoderControlHealthy :=
   "DB_TrolleyCalibrationDiag".qx_EncoderControlHealthy;

   "HMI_DB".Calibration.Trolley.Diagnostics.StartupDataConsistent :=
   "DB_TrolleyCalibrationDiag".qx_StartupDataConsistent;

   "HMI_DB".Calibration.Trolley.Diagnostics.NoMovementWithoutCommand :=
   "DB_TrolleyCalibrationDiag".qx_NoMovementWithoutCommand;

   "HMI_DB".Calibration.Trolley.Diagnostics.NoManualMovementDetected :=
   "DB_TrolleyCalibrationDiag".qx_NoManualMovementDetected;

   "HMI_DB".Calibration.Trolley.Diagnostics.EncoderUpdatesDuringMotion :=
   "DB_TrolleyCalibrationDiag".qx_EncoderUpdatesDuringMotion;

   "HMI_DB".Calibration.Trolley.Diagnostics.EncoderReplacementNotDetected :=
   "DB_TrolleyCalibrationDiag".qx_EncoderReplacementNotDetected;
END_REGION

REGION Network 15: Калібровка механізму крана
END_REGION

REGION Network 16 (SCL): Формування цільової координати у мм для пресету енкодера
   "DB_Calibration".Crane.PresetTargetPosition1_mm :=
   "DB_Calibration".Crane.ReferencePosition_mm
   + "DB_Calibration".Crane.VirtualOffset_mm
   + "DB_Calibration".Crane.TravelAfterReference1_mm;

   "DB_Calibration".Crane.PresetTargetPosition2_mm :=
   "DB_Calibration".Crane.ReferencePosition_mm
   + "DB_Calibration".Crane.VirtualOffset_mm
   + "DB_Calibration".Crane.TravelAfterReference2_mm;
END_REGION

REGION Network 17: Підготовка значення в інкрементах для пресету енкодера 4BR1
   RUNG wire#powerrail
      "FC_PositionToRaw"(Enable := TRUE, Position_mm := "DB_Calibration".Crane.PresetTargetPosition1_mm, RawPoint1 := "DB_EncoderScaling".Enc_4BR1.RawPoint1, PositionPoint1_mm := "DB_EncoderScaling".Enc_4BR1.PositionPoint1_mm, RawPoint2 := "DB_EncoderScaling".Enc_4BR1.RawPoint2, PositionPoint2_mm := "DB_EncoderScaling".Enc_4BR1.PositionPoint2_mm, RawMinimum := DINT#0, RawMaximum := DINT#1073741823, RawPosition => "DB_Calibration".Crane.PresetValueRaw1, RawPositionValid => "DB_Calibration".Crane.PresetValueRaw1Valid, CalculationValid => "DB_Calibration".Crane.PresetCalculation1Valid, ConfigurationValid => "DB_Calibration".Crane.PresetConfiguration1Valid, InConfiguredRange => "DB_Calibration".Crane.Preset1InConfiguredRange, InRawRange => "DB_Calibration".Crane.Preset1InRawRange, Scale_mm_per_count => "DB_Calibration".Crane.PresetScale1_mm_per_count, CalculatedRaw => "DB_Calibration".Crane.PresetCalculatedRaw1, Status => "DB_Calibration".Crane.PresetCalcStatus1)
   END_RUNG
   // the same network as SCL:
   "FC_PositionToRaw"(Enable := TRUE,
                      Position_mm := "DB_Calibration".Crane.PresetTargetPosition1_mm,
                      RawPoint1 := "DB_EncoderScaling".Enc_4BR1.RawPoint1,
                      PositionPoint1_mm := "DB_EncoderScaling".Enc_4BR1.PositionPoint1_mm,
                      RawPoint2 := "DB_EncoderScaling".Enc_4BR1.RawPoint2,
                      PositionPoint2_mm := "DB_EncoderScaling".Enc_4BR1.PositionPoint2_mm,
                      RawMinimum := DINT#0,
                      RawMaximum := DINT#1073741823,
                      RawPosition => "DB_Calibration".Crane.PresetValueRaw1,
                      RawPositionValid => "DB_Calibration".Crane.PresetValueRaw1Valid,
                      CalculationValid => "DB_Calibration".Crane.PresetCalculation1Valid,
                      ConfigurationValid => "DB_Calibration".Crane.PresetConfiguration1Valid,
                      InConfiguredRange => "DB_Calibration".Crane.Preset1InConfiguredRange,
                      InRawRange => "DB_Calibration".Crane.Preset1InRawRange,
                      Scale_mm_per_count => "DB_Calibration".Crane.PresetScale1_mm_per_count,
                      CalculatedRaw => "DB_Calibration".Crane.PresetCalculatedRaw1,
                      Status => "DB_Calibration".Crane.PresetCalcStatus1);
END_REGION

REGION Network 18: Підготовка значення в інкрементах для пресету енкодера 4BR2
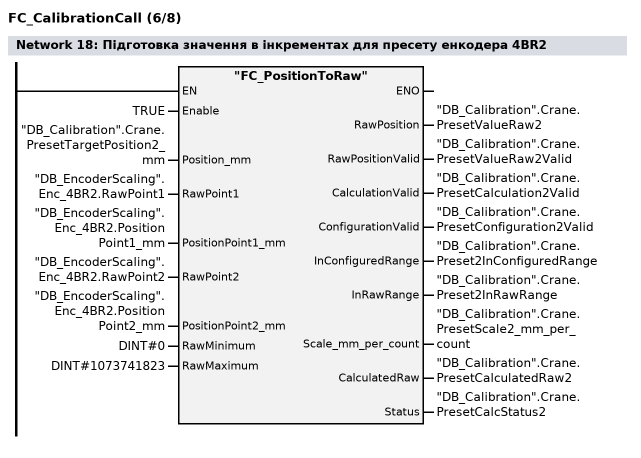
   RUNG wire#powerrail
      "FC_PositionToRaw"(Enable := TRUE, Position_mm := "DB_Calibration".Crane.PresetTargetPosition2_mm, RawPoint1 := "DB_EncoderScaling".Enc_4BR2.RawPoint1, PositionPoint1_mm := "DB_EncoderScaling".Enc_4BR2.PositionPoint1_mm, RawPoint2 := "DB_EncoderScaling".Enc_4BR2.RawPoint2, PositionPoint2_mm := "DB_EncoderScaling".Enc_4BR2.PositionPoint2_mm, RawMinimum := DINT#0, RawMaximum := DINT#1073741823, RawPosition => "DB_Calibration".Crane.PresetValueRaw2, RawPositionValid => "DB_Calibration".Crane.PresetValueRaw2Valid, CalculationValid => "DB_Calibration".Crane.PresetCalculation2Valid, ConfigurationValid => "DB_Calibration".Crane.PresetConfiguration2Valid, InConfiguredRange => "DB_Calibration".Crane.Preset2InConfiguredRange, InRawRange => "DB_Calibration".Crane.Preset2InRawRange, Scale_mm_per_count => "DB_Calibration".Crane.PresetScale2_mm_per_count, CalculatedRaw => "DB_Calibration".Crane.PresetCalculatedRaw2, Status => "DB_Calibration".Crane.PresetCalcStatus2)
   END_RUNG
   // the same network as SCL:
   "FC_PositionToRaw"(Enable := TRUE,
                      Position_mm := "DB_Calibration".Crane.PresetTargetPosition2_mm,
                      RawPoint1 := "DB_EncoderScaling".Enc_4BR2.RawPoint1,
                      PositionPoint1_mm := "DB_EncoderScaling".Enc_4BR2.PositionPoint1_mm,
                      RawPoint2 := "DB_EncoderScaling".Enc_4BR2.RawPoint2,
                      PositionPoint2_mm := "DB_EncoderScaling".Enc_4BR2.PositionPoint2_mm,
                      RawMinimum := DINT#0,
                      RawMaximum := DINT#1073741823,
                      RawPosition => "DB_Calibration".Crane.PresetValueRaw2,
                      RawPositionValid => "DB_Calibration".Crane.PresetValueRaw2Valid,
                      CalculationValid => "DB_Calibration".Crane.PresetCalculation2Valid,
                      ConfigurationValid => "DB_Calibration".Crane.PresetConfiguration2Valid,
                      InConfiguredRange => "DB_Calibration".Crane.Preset2InConfiguredRange,
                      InRawRange => "DB_Calibration".Crane.Preset2InRawRange,
                      Scale_mm_per_count => "DB_Calibration".Crane.PresetScale2_mm_per_count,
                      CalculatedRaw => "DB_Calibration".Crane.PresetCalculatedRaw2,
                      Status => "DB_Calibration".Crane.PresetCalcStatus2);
END_REGION

REGION Network 19: Калібровка енкодерів 4BR1 та 4BR2 механізму моста крана
   // 2026-08-13: Додано умову, що для калібровки крана візок не повинен бути в районі технологічного кінцевика зниження швидкості назад 3К3, а також його відповідного положення по енкодеру
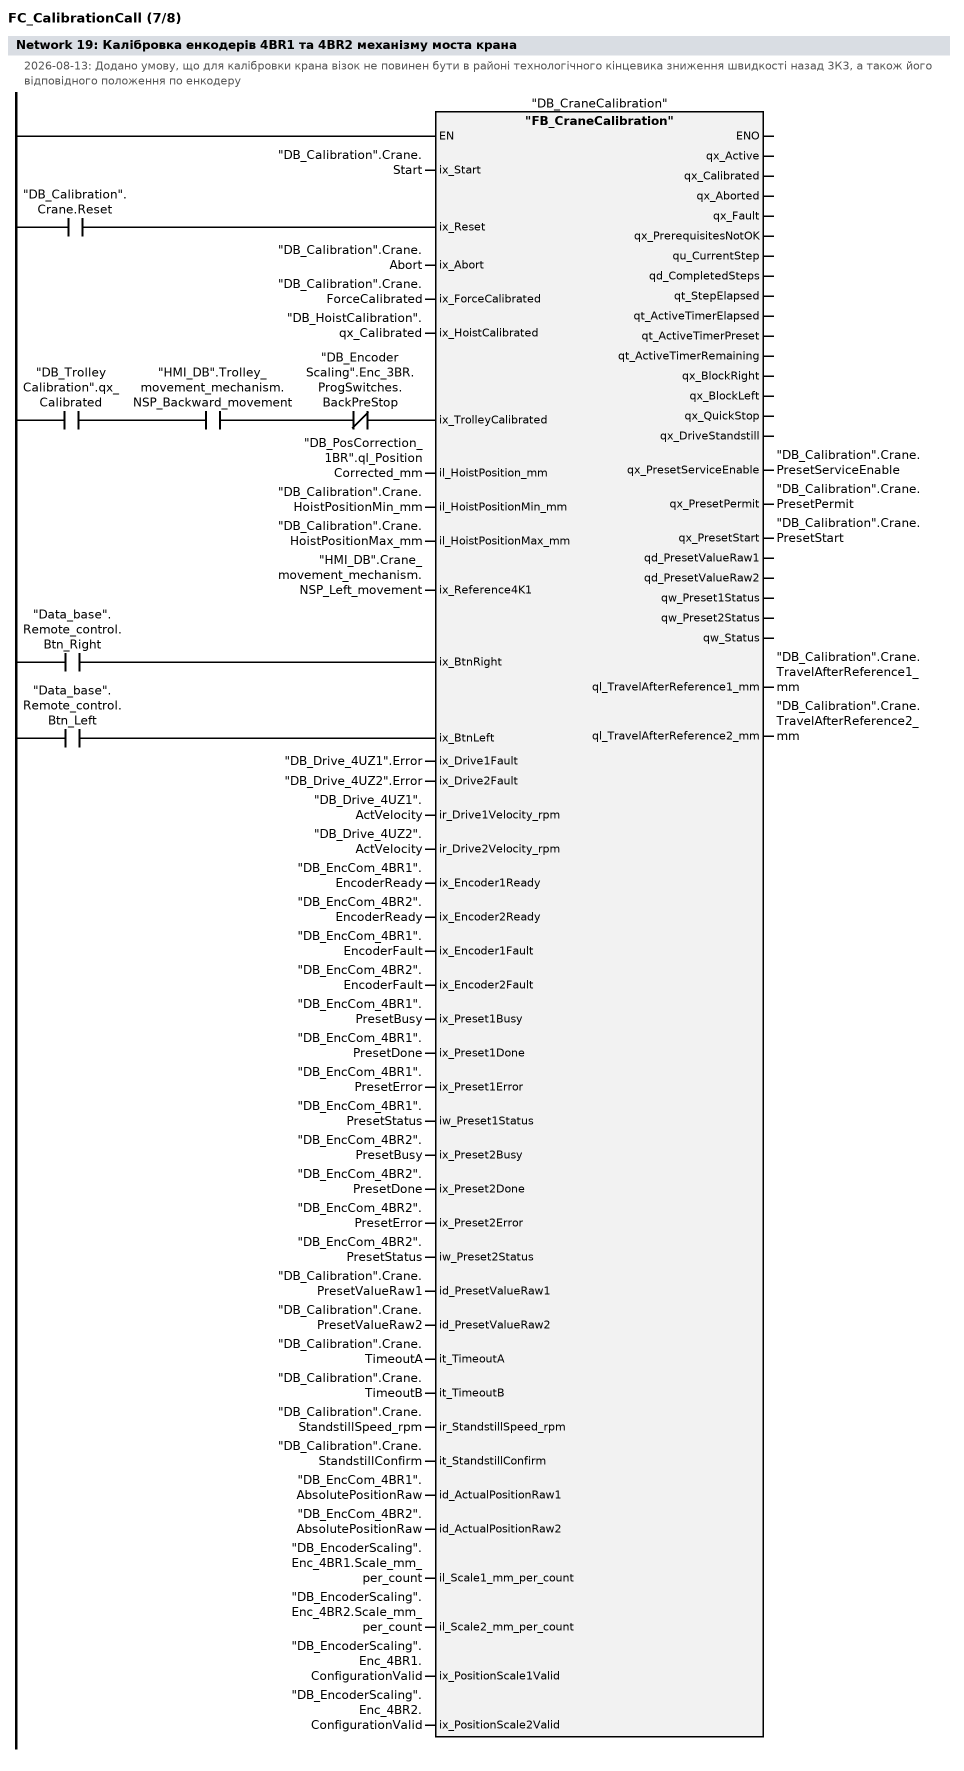
   RUNG wire#powerrail
      "DB_CraneCalibration"(ix_Reset := wire#w1, ix_TrolleyCalibrated := wire#w2, ix_BtnRight := wire#w3, ix_BtnLeft := wire#w4, ix_Start := "DB_Calibration".Crane.Start, ix_Abort := "DB_Calibration".Crane.Abort, ix_ForceCalibrated := "DB_Calibration".Crane.ForceCalibrated, ix_HoistCalibrated := "DB_HoistCalibration".qx_Calibrated, il_HoistPosition_mm := "DB_PosCorrection_1BR".ql_PositionCorrected_mm, il_HoistPositionMin_mm := "DB_Calibration".Crane.HoistPositionMin_mm, il_HoistPositionMax_mm := "DB_Calibration".Crane.HoistPositionMax_mm, ix_Reference4K1 := "HMI_DB".Crane_movement_mechanism.NSP_Left_movement, ix_Drive1Fault := "DB_Drive_4UZ1".Error, ix_Drive2Fault := "DB_Drive_4UZ2".Error, ir_Drive1Velocity_rpm := "DB_Drive_4UZ1".ActVelocity, ir_Drive2Velocity_rpm := "DB_Drive_4UZ2".ActVelocity, ix_Encoder1Ready := "DB_EncCom_4BR1".EncoderReady, ix_Encoder2Ready := "DB_EncCom_4BR2".EncoderReady, ix_Encoder1Fault := "DB_EncCom_4BR1".EncoderFault, ix_Encoder2Fault := "DB_EncCom_4BR2".EncoderFault, ix_Preset1Busy := "DB_EncCom_4BR1".PresetBusy, ix_Preset1Done := "DB_EncCom_4BR1".PresetDone, ix_Preset1Error := "DB_EncCom_4BR1".PresetError, iw_Preset1Status := "DB_EncCom_4BR1".PresetStatus, ix_Preset2Busy := "DB_EncCom_4BR2".PresetBusy, ix_Preset2Done := "DB_EncCom_4BR2".PresetDone, ix_Preset2Error := "DB_EncCom_4BR2".PresetError, iw_Preset2Status := "DB_EncCom_4BR2".PresetStatus, id_PresetValueRaw1 := "DB_Calibration".Crane.PresetValueRaw1, id_PresetValueRaw2 := "DB_Calibration".Crane.PresetValueRaw2, it_TimeoutA := "DB_Calibration".Crane.TimeoutA, it_TimeoutB := "DB_Calibration".Crane.TimeoutB, ir_StandstillSpeed_rpm := "DB_Calibration".Crane.StandstillSpeed_rpm, it_StandstillConfirm := "DB_Calibration".Crane.StandstillConfirm, id_ActualPositionRaw1 := "DB_EncCom_4BR1".AbsolutePositionRaw, id_ActualPositionRaw2 := "DB_EncCom_4BR2".AbsolutePositionRaw, il_Scale1_mm_per_count := "DB_EncoderScaling".Enc_4BR1.Scale_mm_per_count, il_Scale2_mm_per_count := "DB_EncoderScaling".Enc_4BR2.Scale_mm_per_count, ix_PositionScale1Valid := "DB_EncoderScaling".Enc_4BR1.ConfigurationValid, ix_PositionScale2Valid := "DB_EncoderScaling".Enc_4BR2.ConfigurationValid, qx_Active =>, qx_Calibrated =>, qx_Aborted =>, qx_Fault =>, qx_PrerequisitesNotOK =>, qu_CurrentStep =>, qd_CompletedSteps =>, qt_StepElapsed =>, qt_ActiveTimerElapsed =>, qt_ActiveTimerPreset =>, qt_ActiveTimerRemaining =>, qx_BlockRight =>, qx_BlockLeft =>, qx_QuickStop =>, qx_DriveStandstill =>, qx_PresetServiceEnable => "DB_Calibration".Crane.PresetServiceEnable, qx_PresetPermit => "DB_Calibration".Crane.PresetPermit, qx_PresetStart => "DB_Calibration".Crane.PresetStart, qd_PresetValueRaw1 =>, qd_PresetValueRaw2 =>, qw_Preset1Status =>, qw_Preset2Status =>, qw_Status =>, ql_TravelAfterReference1_mm => "DB_Calibration".Crane.TravelAfterReference1_mm, ql_TravelAfterReference2_mm => "DB_Calibration".Crane.TravelAfterReference2_mm)
   END_RUNG
   RUNG wire#powerrail
      Contact( "DB_Calibration".Crane.Reset )
   END_RUNG wire#w1
   RUNG wire#powerrail
      Contact( "DB_TrolleyCalibration".qx_Calibrated )
      Contact( "HMI_DB".Trolley_movement_mechanism.NSP_Backward_movement )
      I_Contact( "DB_EncoderScaling".Enc_3BR.ProgSwitches.BackPreStop )
   END_RUNG wire#w2
   RUNG wire#powerrail
      Contact( "Data_base".Remote_control.Btn_Right )
   END_RUNG wire#w3
   RUNG wire#powerrail
      Contact( "Data_base".Remote_control.Btn_Left )
   END_RUNG wire#w4
   // the same network as SCL:
   "DB_CraneCalibration"(ix_Start := "DB_Calibration".Crane.Start,   // "FB_CraneCalibration"
                         ix_Reset := "DB_Calibration".Crane.Reset,
                         ix_Abort := "DB_Calibration".Crane.Abort,
                         ix_ForceCalibrated := "DB_Calibration".Crane.ForceCalibrated,
                         ix_HoistCalibrated := "DB_HoistCalibration".qx_Calibrated,
                         ix_TrolleyCalibrated := "DB_TrolleyCalibration".qx_Calibrated AND "HMI_DB".Trolley_movement_mechanism.NSP_Backward_movement AND NOT "DB_EncoderScaling".Enc_3BR.ProgSwitches.BackPreStop,
                         il_HoistPosition_mm := "DB_PosCorrection_1BR".ql_PositionCorrected_mm,
                         il_HoistPositionMin_mm := "DB_Calibration".Crane.HoistPositionMin_mm,
                         il_HoistPositionMax_mm := "DB_Calibration".Crane.HoistPositionMax_mm,
                         ix_Reference4K1 := "HMI_DB".Crane_movement_mechanism.NSP_Left_movement,
                         ix_BtnRight := "Data_base".Remote_control.Btn_Right,
                         ix_BtnLeft := "Data_base".Remote_control.Btn_Left,
                         ix_Drive1Fault := "DB_Drive_4UZ1".Error,
                         ix_Drive2Fault := "DB_Drive_4UZ2".Error,
                         ir_Drive1Velocity_rpm := "DB_Drive_4UZ1".ActVelocity,
                         ir_Drive2Velocity_rpm := "DB_Drive_4UZ2".ActVelocity,
                         ix_Encoder1Ready := "DB_EncCom_4BR1".EncoderReady,
                         ix_Encoder2Ready := "DB_EncCom_4BR2".EncoderReady,
                         ix_Encoder1Fault := "DB_EncCom_4BR1".EncoderFault,
                         ix_Encoder2Fault := "DB_EncCom_4BR2".EncoderFault,
                         ix_Preset1Busy := "DB_EncCom_4BR1".PresetBusy,
                         ix_Preset1Done := "DB_EncCom_4BR1".PresetDone,
                         ix_Preset1Error := "DB_EncCom_4BR1".PresetError,
                         iw_Preset1Status := "DB_EncCom_4BR1".PresetStatus,
                         ix_Preset2Busy := "DB_EncCom_4BR2".PresetBusy,
                         ix_Preset2Done := "DB_EncCom_4BR2".PresetDone,
                         ix_Preset2Error := "DB_EncCom_4BR2".PresetError,
                         iw_Preset2Status := "DB_EncCom_4BR2".PresetStatus,
                         id_PresetValueRaw1 := "DB_Calibration".Crane.PresetValueRaw1,
                         id_PresetValueRaw2 := "DB_Calibration".Crane.PresetValueRaw2,
                         it_TimeoutA := "DB_Calibration".Crane.TimeoutA,
                         it_TimeoutB := "DB_Calibration".Crane.TimeoutB,
                         ir_StandstillSpeed_rpm := "DB_Calibration".Crane.StandstillSpeed_rpm,
                         it_StandstillConfirm := "DB_Calibration".Crane.StandstillConfirm,
                         id_ActualPositionRaw1 := "DB_EncCom_4BR1".AbsolutePositionRaw,
                         id_ActualPositionRaw2 := "DB_EncCom_4BR2".AbsolutePositionRaw,
                         il_Scale1_mm_per_count := "DB_EncoderScaling".Enc_4BR1.Scale_mm_per_count,
                         il_Scale2_mm_per_count := "DB_EncoderScaling".Enc_4BR2.Scale_mm_per_count,
                         ix_PositionScale1Valid := "DB_EncoderScaling".Enc_4BR1.ConfigurationValid,
                         ix_PositionScale2Valid := "DB_EncoderScaling".Enc_4BR2.ConfigurationValid,
                         qx_PresetServiceEnable => "DB_Calibration".Crane.PresetServiceEnable,
                         qx_PresetPermit => "DB_Calibration".Crane.PresetPermit,
                         qx_PresetStart => "DB_Calibration".Crane.PresetStart,
                         ql_TravelAfterReference1_mm => "DB_Calibration".Crane.TravelAfterReference1_mm,
                         ql_TravelAfterReference2_mm => "DB_Calibration".Crane.TravelAfterReference2_mm);
END_REGION

REGION Network 20 (SCL): Пресет енкодерів моста 4BR1 та 4BR2
   // Preset control for encoder 4BR1
   "DB_EncCtrl"."4BR1".PresetServiceEnable :=
   "DB_Calibration".Crane.PresetServiceEnable;

   "DB_EncCtrl"."4BR1".PresetPermit :=
   "DB_Calibration".Crane.PresetPermit;

   "DB_EncCtrl"."4BR1".PresetStart :=
   "DB_Calibration".Crane.PresetStart;


   // Preset control for encoder 4BR2
   "DB_EncCtrl"."4BR2".PresetServiceEnable :=
   "DB_Calibration".Crane.PresetServiceEnable;

   "DB_EncCtrl"."4BR2".PresetPermit :=
   "DB_Calibration".Crane.PresetPermit;

   "DB_EncCtrl"."4BR2".PresetStart :=
   "DB_Calibration".Crane.PresetStart;


   // Individual preset values
   "DB_EncCtrl"."4BR1".PresetValueRaw :=
   "DB_CraneCalibration".qd_PresetValueRaw1;

   "DB_EncCtrl"."4BR2".PresetValueRaw :=
   "DB_CraneCalibration".qd_PresetValueRaw2;
END_REGION

REGION Network 21: Діагностика калібровки енкодерів 4BR1 та 4BR2 механізму моста
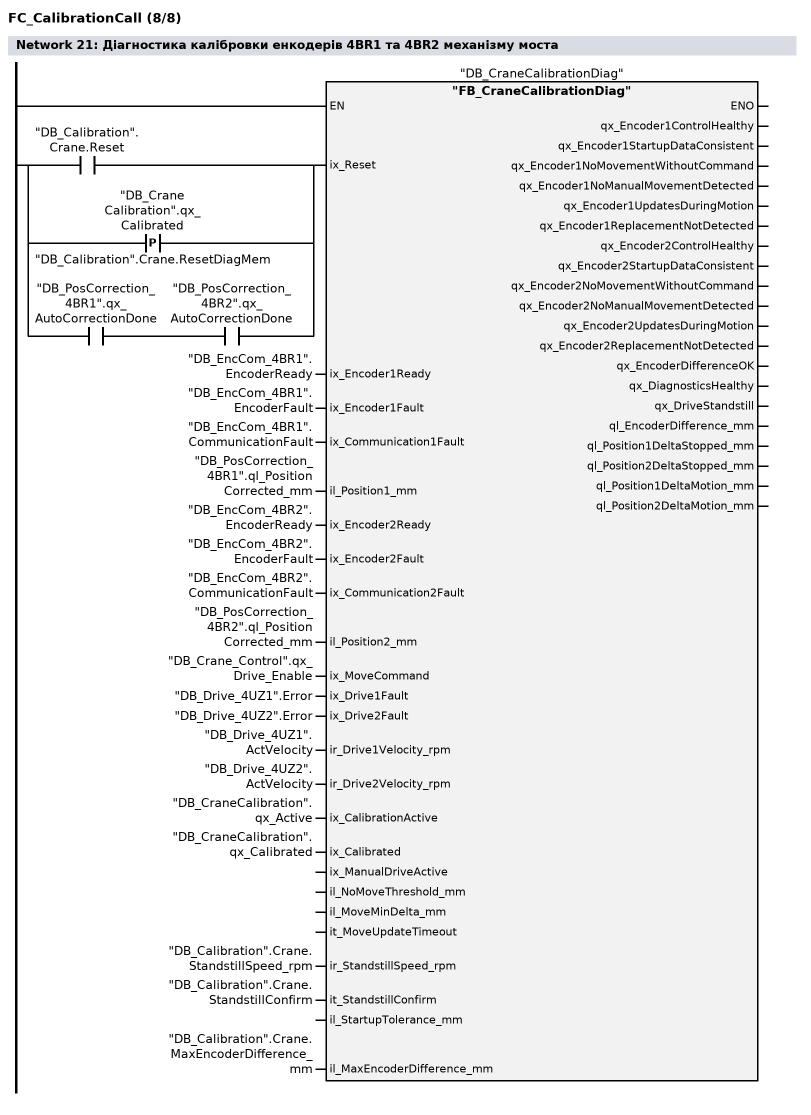
   RUNG wire#powerrail
      "DB_CraneCalibrationDiag"(ix_Reset := wire#w1, ix_Encoder1Ready := "DB_EncCom_4BR1".EncoderReady, ix_Encoder1Fault := "DB_EncCom_4BR1".EncoderFault, ix_Communication1Fault := "DB_EncCom_4BR1".CommunicationFault, il_Position1_mm := "DB_PosCorrection_4BR1".ql_PositionCorrected_mm, ix_Encoder2Ready := "DB_EncCom_4BR2".EncoderReady, ix_Encoder2Fault := "DB_EncCom_4BR2".EncoderFault, ix_Communication2Fault := "DB_EncCom_4BR2".CommunicationFault, il_Position2_mm := "DB_PosCorrection_4BR2".ql_PositionCorrected_mm, ix_MoveCommand := "DB_Crane_Control".qx_Drive_Enable, ix_Drive1Fault := "DB_Drive_4UZ1".Error, ix_Drive2Fault := "DB_Drive_4UZ2".Error, ir_Drive1Velocity_rpm := "DB_Drive_4UZ1".ActVelocity, ir_Drive2Velocity_rpm := "DB_Drive_4UZ2".ActVelocity, ix_CalibrationActive := "DB_CraneCalibration".qx_Active, ix_Calibrated := "DB_CraneCalibration".qx_Calibrated, ix_ManualDriveActive :=, il_NoMoveThreshold_mm :=, il_MoveMinDelta_mm :=, it_MoveUpdateTimeout :=, ir_StandstillSpeed_rpm := "DB_Calibration".Crane.StandstillSpeed_rpm, it_StandstillConfirm := "DB_Calibration".Crane.StandstillConfirm, il_StartupTolerance_mm :=, il_MaxEncoderDifference_mm := "DB_Calibration".Crane.MaxEncoderDifference_mm, qx_Encoder1ControlHealthy =>, qx_Encoder1StartupDataConsistent =>, qx_Encoder1NoMovementWithoutCommand =>, qx_Encoder1NoManualMovementDetected =>, qx_Encoder1UpdatesDuringMotion =>, qx_Encoder1ReplacementNotDetected =>, qx_Encoder2ControlHealthy =>, qx_Encoder2StartupDataConsistent =>, qx_Encoder2NoMovementWithoutCommand =>, qx_Encoder2NoManualMovementDetected =>, qx_Encoder2UpdatesDuringMotion =>, qx_Encoder2ReplacementNotDetected =>, qx_EncoderDifferenceOK =>, qx_DiagnosticsHealthy =>, qx_DriveStandstill =>, ql_EncoderDifference_mm =>, ql_Position1DeltaStopped_mm =>, ql_Position2DeltaStopped_mm =>, ql_Position1DeltaMotion_mm =>, ql_Position2DeltaMotion_mm =>)
   END_RUNG
   RUNG wire#powerrail
      Contact( "DB_Calibration".Crane.Reset )
   END_RUNG wire#w1
   RUNG wire#powerrail
      P_Contact(operand := "DB_CraneCalibration".qx_Calibrated, bit := "DB_Calibration".Crane.ResetDiagMem)
   END_RUNG wire#w1
   RUNG wire#powerrail
      Contact( "DB_PosCorrection_4BR1".qx_AutoCorrectionDone )
      Contact( "DB_PosCorrection_4BR2".qx_AutoCorrectionDone )
   END_RUNG wire#w1
   // the same network as SCL:
   #_w1 := "DB_CraneCalibration".qx_Calibrated AND NOT "DB_Calibration".Crane.ResetDiagMem;   // rising edge of "DB_CraneCalibration".qx_Calibrated
   "DB_Calibration".Crane.ResetDiagMem := "DB_CraneCalibration".qx_Calibrated;
   "DB_CraneCalibrationDiag"(ix_Reset := "DB_Calibration".Crane.Reset OR #_w1 OR ("DB_PosCorrection_4BR1".qx_AutoCorrectionDone AND "DB_PosCorrection_4BR2".qx_AutoCorrectionDone),   // "FB_CraneCalibrationDiag"
                           ix_Encoder1Ready := "DB_EncCom_4BR1".EncoderReady,
                           ix_Encoder1Fault := "DB_EncCom_4BR1".EncoderFault,
                           ix_Communication1Fault := "DB_EncCom_4BR1".CommunicationFault,
                           il_Position1_mm := "DB_PosCorrection_4BR1".ql_PositionCorrected_mm,
                           ix_Encoder2Ready := "DB_EncCom_4BR2".EncoderReady,
                           ix_Encoder2Fault := "DB_EncCom_4BR2".EncoderFault,
                           ix_Communication2Fault := "DB_EncCom_4BR2".CommunicationFault,
                           il_Position2_mm := "DB_PosCorrection_4BR2".ql_PositionCorrected_mm,
                           ix_MoveCommand := "DB_Crane_Control".qx_Drive_Enable,
                           ix_Drive1Fault := "DB_Drive_4UZ1".Error,
                           ix_Drive2Fault := "DB_Drive_4UZ2".Error,
                           ir_Drive1Velocity_rpm := "DB_Drive_4UZ1".ActVelocity,
                           ir_Drive2Velocity_rpm := "DB_Drive_4UZ2".ActVelocity,
                           ix_CalibrationActive := "DB_CraneCalibration".qx_Active,
                           ix_Calibrated := "DB_CraneCalibration".qx_Calibrated,
                           ir_StandstillSpeed_rpm := "DB_Calibration".Crane.StandstillSpeed_rpm,
                           it_StandstillConfirm := "DB_Calibration".Crane.StandstillConfirm,
                           il_MaxEncoderDifference_mm := "DB_Calibration".Crane.MaxEncoderDifference_mm);
END_REGION

REGION Network 22 (SCL): Калібровка моста - дані на візуалізацію
   // ============================================================
   // HMI mapping - crane calibration
   // ============================================================

   // Main calibration state
   "HMI_DB".Calibration.Crane.Active :=
   "DB_CraneCalibration".qx_Active;

   "HMI_DB".Calibration.Crane.Calibrated :=
   "DB_CraneCalibration".qx_Calibrated;

   "HMI_DB".Calibration.Crane.Fault :=
   "DB_CraneCalibration".qx_Fault;

   "HMI_DB".Calibration.Crane.Aborted :=
   "DB_CraneCalibration".qx_Aborted;

   "HMI_DB".Calibration.Crane.PrerequisitesNotOK :=
   "DB_CraneCalibration".qx_PrerequisitesNotOK;

   "HMI_DB".Calibration.Crane.CurrentStep :=
   "DB_CraneCalibration".qu_CurrentStep;

   "HMI_DB".Calibration.Crane.CompletedSteps :=
   "DB_CraneCalibration".qd_CompletedSteps;


   // Reference switch 4K1
   "HMI_DB".Calibration.Crane.Reference4K1 :=
   "DB_CraneCalibration".ix_Reference4K1;


   // Encoder positions
   "HMI_DB".Calibration.Crane.Position4BR1_mm :=
   "DB_PosCorrection_4BR1".qd_PositionCorrectedRounded_mm;

   "HMI_DB".Calibration.Crane.Position4BR2_mm :=
   "DB_PosCorrection_4BR2".qd_PositionCorrectedRounded_mm;

   // Actual drive velocities
   "HMI_DB".Calibration.Crane.Drive1Velocity_rpm :=
   "DB_Drive_4UZ1".ActVelocity;

   "HMI_DB".Calibration.Crane.Drive2Velocity_rpm :=
   "DB_Drive_4UZ2".ActVelocity;


   // Active calibration timer
   "HMI_DB".Calibration.Crane.TimerRemaining :=
   "DB_CraneCalibration".qt_ActiveTimerRemaining;

   // ============================================================
   // HMI mapping - crane calibration timer
   // ============================================================

   #TempRemainingSeconds :=
   TIME_TO_UDINT("DB_CraneCalibration".qt_ActiveTimerRemaining)
   / UDINT#1000;

   "HMI_DB".Calibration.Crane.TimerRemaining_Min :=
   UDINT_TO_UINT(
                 #TempRemainingSeconds / UDINT#60
   );

   "HMI_DB".Calibration.Crane.TimerRemaining_Sec :=
   UDINT_TO_UINT(
                 #TempRemainingSeconds MOD UDINT#60
   );


   // ============================================================
   // HMI mapping - crane completed calibration steps
   // ============================================================

   "HMI_DB".Calibration.Crane.Steps_Completed.Step10 :=
   "DB_CraneCalibration".qd_CompletedSteps.%X0;

   "HMI_DB".Calibration.Crane.Steps_Completed.Step20 :=
   "DB_CraneCalibration".qd_CompletedSteps.%X1;

   "HMI_DB".Calibration.Crane.Steps_Completed.Step30 :=
   "DB_CraneCalibration".qd_CompletedSteps.%X2;

   "HMI_DB".Calibration.Crane.Steps_Completed.Step40 :=
   "DB_CraneCalibration".qd_CompletedSteps.%X3;

   "HMI_DB".Calibration.Crane.Steps_Completed.Step50 :=
   "DB_CraneCalibration".qd_CompletedSteps.%X4;

   "HMI_DB".Calibration.Crane.Steps_Completed.Step60 :=
   "DB_CraneCalibration".qd_CompletedSteps.%X5;

   "HMI_DB".Calibration.Crane.Steps_Completed.Step70 :=
   "DB_CraneCalibration".qd_CompletedSteps.%X6;

   "HMI_DB".Calibration.Crane.Steps_Completed.Step80 :=
   "DB_CraneCalibration".qd_CompletedSteps.%X7;

   "HMI_DB".Calibration.Crane.Steps_Completed.Step90 :=
   "DB_CraneCalibration".qd_CompletedSteps.%X8;

   "HMI_DB".Calibration.Crane.Steps_Completed.Step100 :=
   "DB_CraneCalibration".qd_CompletedSteps.%X9;

   "HMI_DB".Calibration.Crane.Steps_Completed.Step110 :=
   "DB_CraneCalibration".qd_CompletedSteps.%X10;

   "HMI_DB".Calibration.Crane.Steps_Completed.Step120 :=
   "DB_CraneCalibration".qd_CompletedSteps.%X11;

   "HMI_DB".Calibration.Crane.Steps_Completed.Step130 :=
   "DB_CraneCalibration".qd_CompletedSteps.%X12;

   // ============================================================
   // HMI mapping - crane active calibration steps
   // ============================================================

   "HMI_DB".Calibration.Crane.Steps_Active.Step10 :=
   "HMI_DB".Calibration.Crane.CurrentStep = UINT#10;

   "HMI_DB".Calibration.Crane.Steps_Active.Step20 :=
   "HMI_DB".Calibration.Crane.CurrentStep = UINT#20;

   "HMI_DB".Calibration.Crane.Steps_Active.Step30 :=
   "HMI_DB".Calibration.Crane.CurrentStep = UINT#30;

   "HMI_DB".Calibration.Crane.Steps_Active.Step40 :=
   "HMI_DB".Calibration.Crane.CurrentStep = UINT#40;

   "HMI_DB".Calibration.Crane.Steps_Active.Step50 :=
   "HMI_DB".Calibration.Crane.CurrentStep = UINT#50;

   "HMI_DB".Calibration.Crane.Steps_Active.Step60 :=
   "HMI_DB".Calibration.Crane.CurrentStep = UINT#60;

   "HMI_DB".Calibration.Crane.Steps_Active.Step70 :=
   "HMI_DB".Calibration.Crane.CurrentStep = UINT#70;

   "HMI_DB".Calibration.Crane.Steps_Active.Step80 :=
   "HMI_DB".Calibration.Crane.CurrentStep = UINT#80;

   "HMI_DB".Calibration.Crane.Steps_Active.Step90 :=
   "HMI_DB".Calibration.Crane.CurrentStep = UINT#90;

   "HMI_DB".Calibration.Crane.Steps_Active.Step100 :=
   "HMI_DB".Calibration.Crane.CurrentStep = UINT#100;

   "HMI_DB".Calibration.Crane.Steps_Active.Step110 :=
   "HMI_DB".Calibration.Crane.CurrentStep = UINT#110;

   "HMI_DB".Calibration.Crane.Steps_Active.Step120 :=
   "HMI_DB".Calibration.Crane.CurrentStep = UINT#120;

   "HMI_DB".Calibration.Crane.Steps_Active.Step130 :=
   "HMI_DB".Calibration.Crane.CurrentStep = UINT#130;

   // ============================================================
   // HMI mapping - crane calibration diagnostics
   // ============================================================

   // Encoder 4BR1
   "HMI_DB".Calibration.Crane.Diagnostics.Encoder1ControlHealthy :=
   "DB_CraneCalibrationDiag".qx_Encoder1ControlHealthy;

   "HMI_DB".Calibration.Crane.Diagnostics.Encoder1StartupDataConsistent :=
   "DB_CraneCalibrationDiag".qx_Encoder1StartupDataConsistent;

   "HMI_DB".Calibration.Crane.Diagnostics.Encoder1NoMovementWithoutCommand :=
   "DB_CraneCalibrationDiag".qx_Encoder1NoMovementWithoutCommand;

   "HMI_DB".Calibration.Crane.Diagnostics.Encoder1NoManualMovementDetected :=
   "DB_CraneCalibrationDiag".qx_Encoder1NoManualMovementDetected;

   "HMI_DB".Calibration.Crane.Diagnostics.Encoder1UpdatesDuringMotion :=
   "DB_CraneCalibrationDiag".qx_Encoder1UpdatesDuringMotion;

   "HMI_DB".Calibration.Crane.Diagnostics.Encoder1ReplacementNotDetected :=
   "DB_CraneCalibrationDiag".qx_Encoder1ReplacementNotDetected;


   // Encoder 4BR2
   "HMI_DB".Calibration.Crane.Diagnostics.Encoder2ControlHealthy :=
   "DB_CraneCalibrationDiag".qx_Encoder2ControlHealthy;

   "HMI_DB".Calibration.Crane.Diagnostics.Encoder2StartupDataConsistent :=
   "DB_CraneCalibrationDiag".qx_Encoder2StartupDataConsistent;

   "HMI_DB".Calibration.Crane.Diagnostics.Encoder2NoMovementWithoutCommand :=
   "DB_CraneCalibrationDiag".qx_Encoder2NoMovementWithoutCommand;

   "HMI_DB".Calibration.Crane.Diagnostics.Encoder2NoManualMovementDetected :=
   "DB_CraneCalibrationDiag".qx_Encoder2NoManualMovementDetected;

   "HMI_DB".Calibration.Crane.Diagnostics.Encoder2UpdatesDuringMotion :=
   "DB_CraneCalibrationDiag".qx_Encoder2UpdatesDuringMotion;

   "HMI_DB".Calibration.Crane.Diagnostics.Encoder2ReplacementNotDetected :=
   "DB_CraneCalibrationDiag".qx_Encoder2ReplacementNotDetected;


   // Encoder difference
   "HMI_DB".Calibration.Crane.Diagnostics.EncoderDifferenceOK :=
   "DB_CraneCalibrationDiag".qx_EncoderDifferenceOK;


   // General diagnostic state
   "HMI_DB".Calibration.Crane.Diagnostics.DiagnosticsHealthy :=
   "DB_CraneCalibrationDiag".qx_DiagnosticsHealthy;

   "HMI_DB".Calibration.Crane.Diagnostics.DriveStandstill :=
   "DB_CraneCalibrationDiag".qx_DriveStandstill;


   // Service values
   "HMI_DB".Calibration.Crane.Diagnostics.EncoderDifference_mm :=
   "DB_CraneCalibrationDiag".ql_EncoderDifference_mm;

   "HMI_DB".Calibration.Crane.Diagnostics.Position1DeltaStopped_mm :=
   "DB_CraneCalibrationDiag".ql_Position1DeltaStopped_mm;

   "HMI_DB".Calibration.Crane.Diagnostics.Position2DeltaStopped_mm :=
   "DB_CraneCalibrationDiag".ql_Position2DeltaStopped_mm;

   "HMI_DB".Calibration.Crane.Diagnostics.Position1DeltaMotion_mm :=
   "DB_CraneCalibrationDiag".ql_Position1DeltaMotion_mm;

   "HMI_DB".Calibration.Crane.Diagnostics.Position2DeltaMotion_mm :=
   "DB_CraneCalibrationDiag".ql_Position2DeltaMotion_mm;
END_REGION
END_FUNCTION

FUNCTION "FC_PositionToRaw" : Void   // FC707, SCL
{ S7_Optimized_Access := 'TRUE' }
VERSION : 0.1
   VAR_INPUT
      Enable : Bool;   // Загальний дозвіл роботи функції
      Position_mm : LReal;   // Цільова координата для перетворення у raw
      RawPoint1 : DInt;   // Raw першої контрольної точки
      PositionPoint1_mm : LReal;   // Координата першої контрольної точки
      RawPoint2 : DInt;   // Raw другої контрольної точки
      PositionPoint2_mm : LReal;   // Координата другої контрольної точки
      RawMinimum : DInt;   // Мінімально допустиме raw
      RawMaximum : DInt;   // Максимально допустиме raw
   END_VAR
   VAR_OUTPUT
      RawPosition : DInt;   // Розраховане raw-значення
      RawPositionValid : Bool;   // Raw можна використовувати для preset
      CalculationValid : Bool;   // Розрахунок виконаний
      ConfigurationValid : Bool;   // Контрольні точки задані коректно
      InConfiguredRange : Bool;   // Position знаходиться між двома контрольними точками
      InRawRange : Bool;   // Результат знаходиться у допустимому raw-діапазоні
      Scale_mm_per_count : LReal;   // Масштаб мм/count
      CalculatedRaw : LReal;   // Розраховане raw до перетворення в DINT
      Status : Word;   // Діагностичне слово
   END_VAR
   VAR_TEMP
      RawSpan : LReal;
      PositionSpan_mm : LReal;
      PositionDelta_mm : LReal;
      PositionMinimum_mm : LReal;
      PositionMaximum_mm : LReal;
   END_VAR
BEGIN
   // ============================================================
   // FC_PositionToRaw
   //
   // Перетворення координати механізму в мм
   // у сире значення енкодера (raw counts).
   //
   // Функція є зворотною до FC_EncoderScale.
   //
   // Для розрахунку використовуються дві контрольні точки:
   //
   // RawPoint1 <-> PositionPoint1_mm
   // RawPoint2 <-> PositionPoint2_mm
   //
   // Position_mm повинна вже містити всі необхідні зміщення.
   // Функція самостійно не розраховує VirtualOffset
   // або інші корекції координати.
   //
   // Якщо Position_mm знаходиться поза діапазоном двох
   // контрольних точок, розрахунок продовжується методом
   // лінійної екстраполяції.
   //
   // Остаточним обмеженням є допустимий raw-діапазон
   // RawMinimum ... RawMaximum.
   // ============================================================


   // ============================================================
   // 1. Початкові значення виходів
   // ============================================================

   #RawPosition := DINT#0;

   #RawPositionValid := FALSE;
   #CalculationValid := FALSE;
   #ConfigurationValid := FALSE;

   #InConfiguredRange := FALSE;
   #InRawRange := FALSE;

   #Scale_mm_per_count := 0.0;
   #CalculatedRaw := 0.0;

   #Status := W#16#0000;

   #RawSpan := 0.0;
   #PositionSpan_mm := 0.0;
   #PositionDelta_mm := 0.0;

   #PositionMinimum_mm := 0.0;
   #PositionMaximum_mm := 0.0;


   // ============================================================
   // 2. Перевірка дозволу роботи функції
   // ============================================================

   IF NOT #Enable THEN

       // Bit 0:
       // Функція вимкнена.
       #Status := #Status OR W#16#0001;

       RETURN;

   END_IF;


   // ============================================================
   // 3. Перевірка raw-точок масштабування
   // ============================================================

   IF #RawPoint1 = #RawPoint2 THEN

       // Bit 1:
       // Raw-значення двох контрольних точок однакові.
       // Розрахунок масштабу неможливий.
       #Status := #Status OR W#16#0002;

       RETURN;

   END_IF;


   // ============================================================
   // 4. Перевірка координат контрольних точок
   // ============================================================

   IF #PositionPoint1_mm = #PositionPoint2_mm THEN

       // Bit 2:
       // Координати двох контрольних точок однакові.
       // Розрахунок масштабу неможливий.
       #Status := #Status OR W#16#0004;

       RETURN;

   END_IF;


   // ============================================================
   // 5. Перевірка допустимого raw-діапазону
   // ============================================================

   IF #RawMinimum >= #RawMaximum THEN

       // Bit 3:
       // Мінімальна та максимальна межі raw задані некоректно.
       #Status := #Status OR W#16#0008;

       RETURN;

   END_IF;


   // ============================================================
   // 6. Конфігурація коректна
   // ============================================================

   #ConfigurationValid := TRUE;

   // Bit 6:
   // Контрольні точки та raw-діапазон задані коректно.
   #Status := #Status OR W#16#0040;


   // ============================================================
   // 7. Розрахунок масштабу
   // ============================================================

   // Перетворення у LREAL виконується до віднімання,
   // щоб уникнути переповнення DINT.

   #RawSpan :=
   DINT_TO_LREAL(#RawPoint2)
   - DINT_TO_LREAL(#RawPoint1);

   #PositionSpan_mm :=
   #PositionPoint2_mm
   - #PositionPoint1_mm;

   #Scale_mm_per_count :=
   #PositionSpan_mm
   / #RawSpan;


   // ============================================================
   // 8. Визначення діапазону між контрольними точками
   // ============================================================

   IF #PositionPoint1_mm <= #PositionPoint2_mm THEN

       #PositionMinimum_mm :=
       #PositionPoint1_mm;

       #PositionMaximum_mm :=
       #PositionPoint2_mm;

   ELSE

       #PositionMinimum_mm :=
       #PositionPoint2_mm;

       #PositionMaximum_mm :=
       #PositionPoint1_mm;

   END_IF;


